REGION Network 40: [Job]Transfer P&P Left Select Job [to Hipot&Thinkness]
   // Configure here when the jobs of the sequence should be started. More jobs could be added.
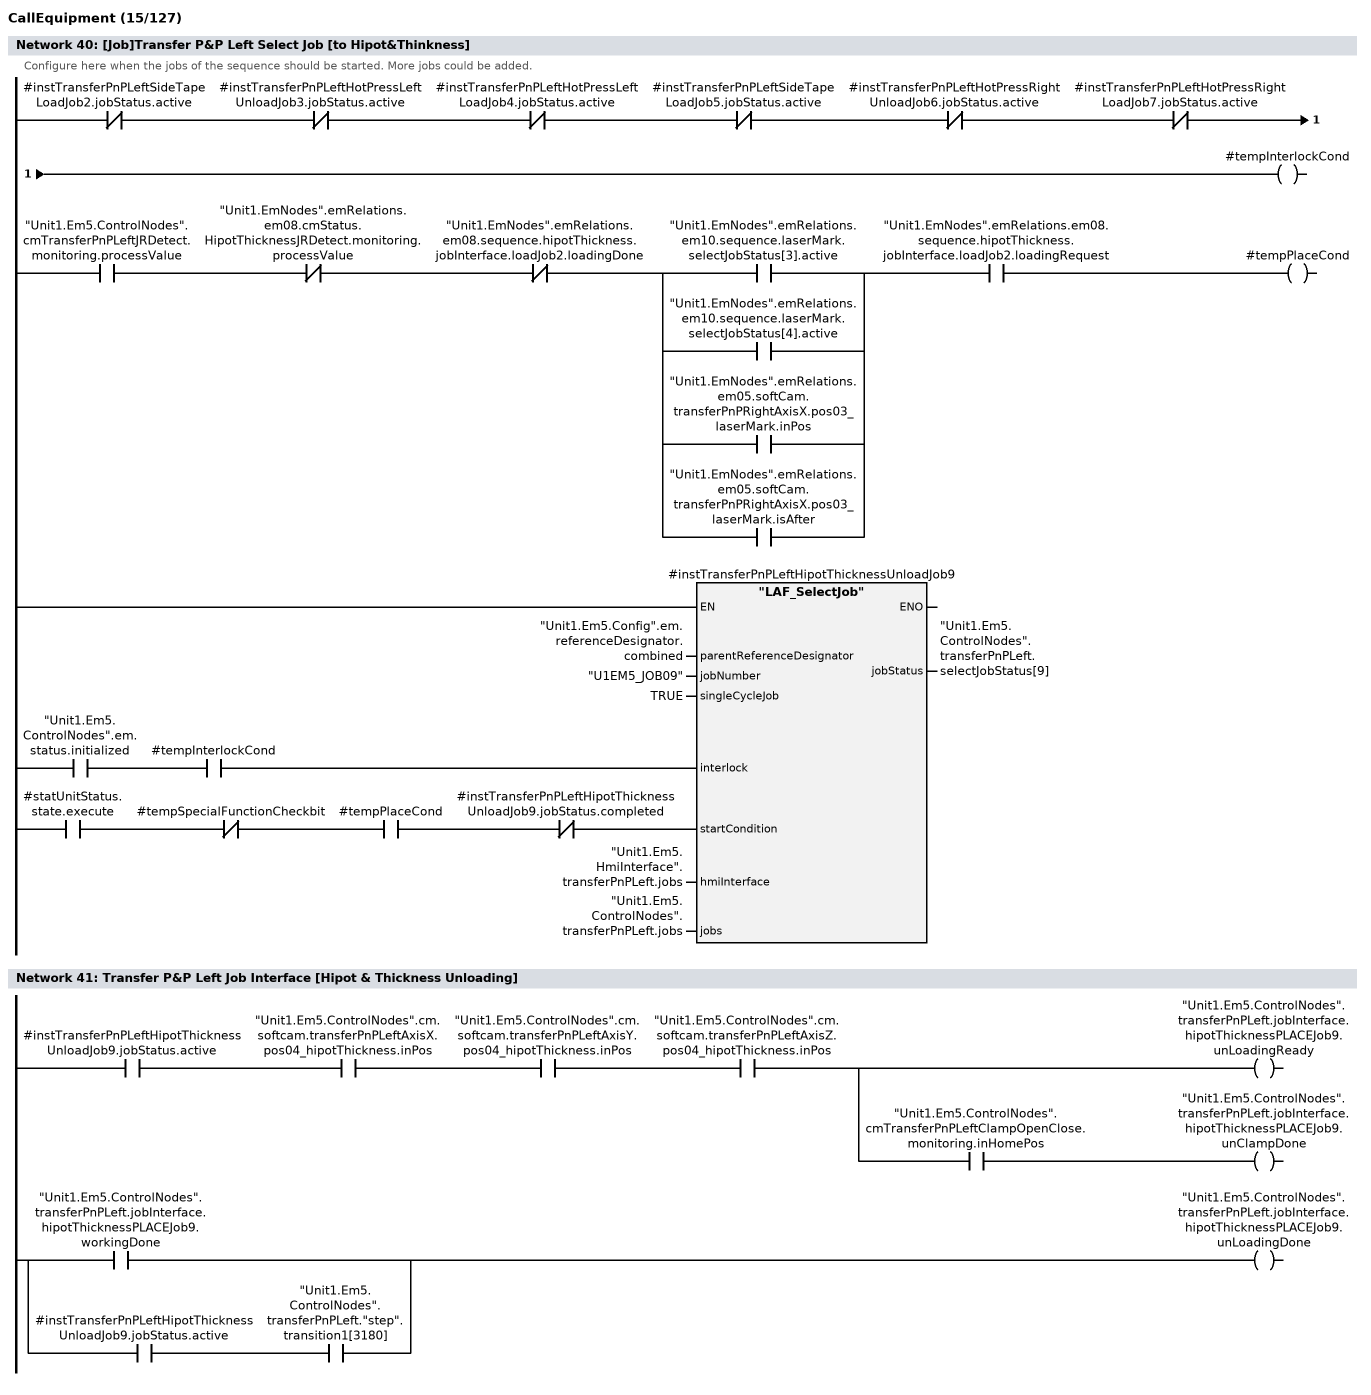
   RUNG wire#powerrail
      I_Contact( #instTransferPnPLeftSideTapeLoadJob2.jobStatus.active )
      I_Contact( #instTransferPnPLeftHotPressLeftUnloadJob3.jobStatus.active )
      I_Contact( #instTransferPnPLeftHotPressLeftLoadJob4.jobStatus.active )
      I_Contact( #instTransferPnPLeftSideTapeLoadJob5.jobStatus.active )
      I_Contact( #instTransferPnPLeftHotPressRightUnloadJob6.jobStatus.active )
      I_Contact( #instTransferPnPLeftHotPressRightLoadJob7.jobStatus.active )
      Coil( #tempInterlockCond )
   END_RUNG
   RUNG wire#powerrail
      Contact( "Unit1.Em5.ControlNodes".cmTransferPnPLeftJRDetect.monitoring.processValue )
      I_Contact( "Unit1.EmNodes".emRelations.em08.cmStatus.HipotThicknessJRDetect.monitoring.processValue )
      I_Contact( "Unit1.EmNodes".emRelations.em08.sequence.hipotThickness.jobInterface.loadJob2.loadingDone )
      wire#w1
      Contact( "Unit1.EmNodes".emRelations.em10.sequence.laserMark.selectJobStatus[3].active )
      wire#w2
      Contact( "Unit1.EmNodes".emRelations.em08.sequence.hipotThickness.jobInterface.loadJob2.loadingRequest )
      Coil( #tempPlaceCond )
   END_RUNG
   RUNG wire#w1
      Contact( "Unit1.EmNodes".emRelations.em10.sequence.laserMark.selectJobStatus[4].active )
   END_RUNG wire#w2
   RUNG wire#w1
      Contact( "Unit1.EmNodes".emRelations.em05.softCam.transferPnPRightAxisX.pos03_laserMark.inPos )
   END_RUNG wire#w2
   RUNG wire#w1
      Contact( "Unit1.EmNodes".emRelations.em05.softCam.transferPnPRightAxisX.pos03_laserMark.isAfter )
   END_RUNG wire#w2
   RUNG wire#powerrail
      #instTransferPnPLeftHipotThicknessUnloadJob9(interlock := wire#w3, startCondition := wire#w4, parentReferenceDesignator := "Unit1.Em5.Config".em.referenceDesignator.combined, jobNumber := "U1EM5_JOB09", singleCycleJob := TRUE, hmiInterface := "Unit1.Em5.HmiInterface".transferPnPLeft.jobs, jobs := "Unit1.Em5.ControlNodes".transferPnPLeft.jobs, jobStatus => "Unit1.Em5.ControlNodes".transferPnPLeft.selectJobStatus[9])
   END_RUNG
   RUNG wire#powerrail
      Contact( "Unit1.Em5.ControlNodes".em.status.initialized )
      Contact( #tempInterlockCond )
   END_RUNG wire#w3
   RUNG wire#powerrail
      Contact( #statUnitStatus.state.execute )
      I_Contact( #tempSpecialFunctionCheckbit )
      Contact( #tempPlaceCond )
      I_Contact( #instTransferPnPLeftHipotThicknessUnloadJob9.jobStatus.completed )
   END_RUNG wire#w4
   // the same network as SCL:
   #tempInterlockCond := NOT #instTransferPnPLeftSideTapeLoadJob2.jobStatus.active AND NOT #instTransferPnPLeftHotPressLeftUnloadJob3.jobStatus.active AND NOT #instTransferPnPLeftHotPressLeftLoadJob4.jobStatus.active AND NOT #instTransferPnPLeftSideTapeLoadJob5.jobStatus.active AND NOT #instTransferPnPLeftHotPressRightUnloadJob6.jobStatus.active AND NOT #instTransferPnPLeftHotPressRightLoadJob7.jobStatus.active;
   #tempPlaceCond := "Unit1.Em5.ControlNodes".cmTransferPnPLeftJRDetect.monitoring.processValue AND NOT "Unit1.EmNodes".emRelations.em08.cmStatus.HipotThicknessJRDetect.monitoring.processValue AND NOT "Unit1.EmNodes".emRelations.em08.sequence.hipotThickness.jobInterface.loadJob2.loadingDone AND ("Unit1.EmNodes".emRelations.em10.sequence.laserMark.selectJobStatus[3].active OR "Unit1.EmNodes".emRelations.em10.sequence.laserMark.selectJobStatus[4].active OR "Unit1.EmNodes".emRelations.em05.softCam.transferPnPRightAxisX.pos03_laserMark.inPos OR "Unit1.EmNodes".emRelations.em05.softCam.transferPnPRightAxisX.pos03_laserMark.isAfter) AND "Unit1.EmNodes".emRelations.em08.sequence.hipotThickness.jobInterface.loadJob2.loadingRequest;
   #instTransferPnPLeftHipotThicknessUnloadJob9(parentReferenceDesignator := "Unit1.Em5.Config".em.referenceDesignator.combined,   // "LAF_SelectJob"
                           jobNumber := "U1EM5_JOB09",
                           singleCycleJob := TRUE,
                           interlock := "Unit1.Em5.ControlNodes".em.status.initialized AND #tempInterlockCond,
                           startCondition := #statUnitStatus.state.execute AND NOT #tempSpecialFunctionCheckbit AND #tempPlaceCond AND NOT #instTransferPnPLeftHipotThicknessUnloadJob9.jobStatus.completed,
                           hmiInterface := "Unit1.Em5.HmiInterface".transferPnPLeft.jobs,
                           jobs := "Unit1.Em5.ControlNodes".transferPnPLeft.jobs,
                           jobStatus => "Unit1.Em5.ControlNodes".transferPnPLeft.selectJobStatus[9]);
END_REGION

REGION Network 41: Transfer P&P Left Job Interface [Hipot & Thickness Unloading]
   RUNG wire#powerrail
      Contact( #instTransferPnPLeftHipotThicknessUnloadJob9.jobStatus.active )
      Contact( "Unit1.Em5.ControlNodes".cm.softcam.transferPnPLeftAxisX.pos04_hipotThickness.inPos )
      Contact( "Unit1.Em5.ControlNodes".cm.softcam.transferPnPLeftAxisY.pos04_hipotThickness.inPos )
      Contact( "Unit1.Em5.ControlNodes".cm.softcam.transferPnPLeftAxisZ.pos04_hipotThickness.inPos )
      wire#w1
      Coil( "Unit1.Em5.ControlNodes".transferPnPLeft.jobInterface.hipotThicknessPLACEJob9.unLoadingReady )
   END_RUNG
   RUNG wire#w1
      Contact( "Unit1.Em5.ControlNodes".cmTransferPnPLeftClampOpenClose.monitoring.inHomePos )
      Coil( "Unit1.Em5.ControlNodes".transferPnPLeft.jobInterface.hipotThicknessPLACEJob9.unClampDone )
   END_RUNG
   RUNG wire#powerrail
      Contact( "Unit1.Em5.ControlNodes".transferPnPLeft.jobInterface.hipotThicknessPLACEJob9.workingDone )
      wire#w2
      Coil( "Unit1.Em5.ControlNodes".transferPnPLeft.jobInterface.hipotThicknessPLACEJob9.unLoadingDone )
   END_RUNG
   RUNG wire#powerrail
      Contact( #instTransferPnPLeftHipotThicknessUnloadJob9.jobStatus.active )
      Contact( "Unit1.Em5.ControlNodes".transferPnPLeft."step".transition1[3180] )
   END_RUNG wire#w2
   // the same network as SCL:
   "Unit1.Em5.ControlNodes".transferPnPLeft.jobInterface.hipotThicknessPLACEJob9.unLoadingReady := #instTransferPnPLeftHipotThicknessUnloadJob9.jobStatus.active AND "Unit1.Em5.ControlNodes".cm.softcam.transferPnPLeftAxisX.pos04_hipotThickness.inPos AND "Unit1.Em5.ControlNodes".cm.softcam.transferPnPLeftAxisY.pos04_hipotThickness.inPos AND "Unit1.Em5.ControlNodes".cm.softcam.transferPnPLeftAxisZ.pos04_hipotThickness.inPos;
   "Unit1.Em5.ControlNodes".transferPnPLeft.jobInterface.hipotThicknessPLACEJob9.unClampDone := "Unit1.Em5.ControlNodes".transferPnPLeft.jobInterface.hipotThicknessPLACEJob9.unLoadingReady AND "Unit1.Em5.ControlNodes".cmTransferPnPLeftClampOpenClose.monitoring.inHomePos;
   "Unit1.Em5.ControlNodes".transferPnPLeft.jobInterface.hipotThicknessPLACEJob9.unLoadingDone := "Unit1.Em5.ControlNodes".transferPnPLeft.jobInterface.hipotThicknessPLACEJob9.workingDone OR (#instTransferPnPLeftHipotThicknessUnloadJob9.jobStatus.active AND "Unit1.Em5.ControlNodes".transferPnPLeft."step".transition1[3180]);
END_REGION

REGION Network 42: Transfer P&P Left Job Interface Working Done [HotPress Left/Right → Hipot&Thickness]
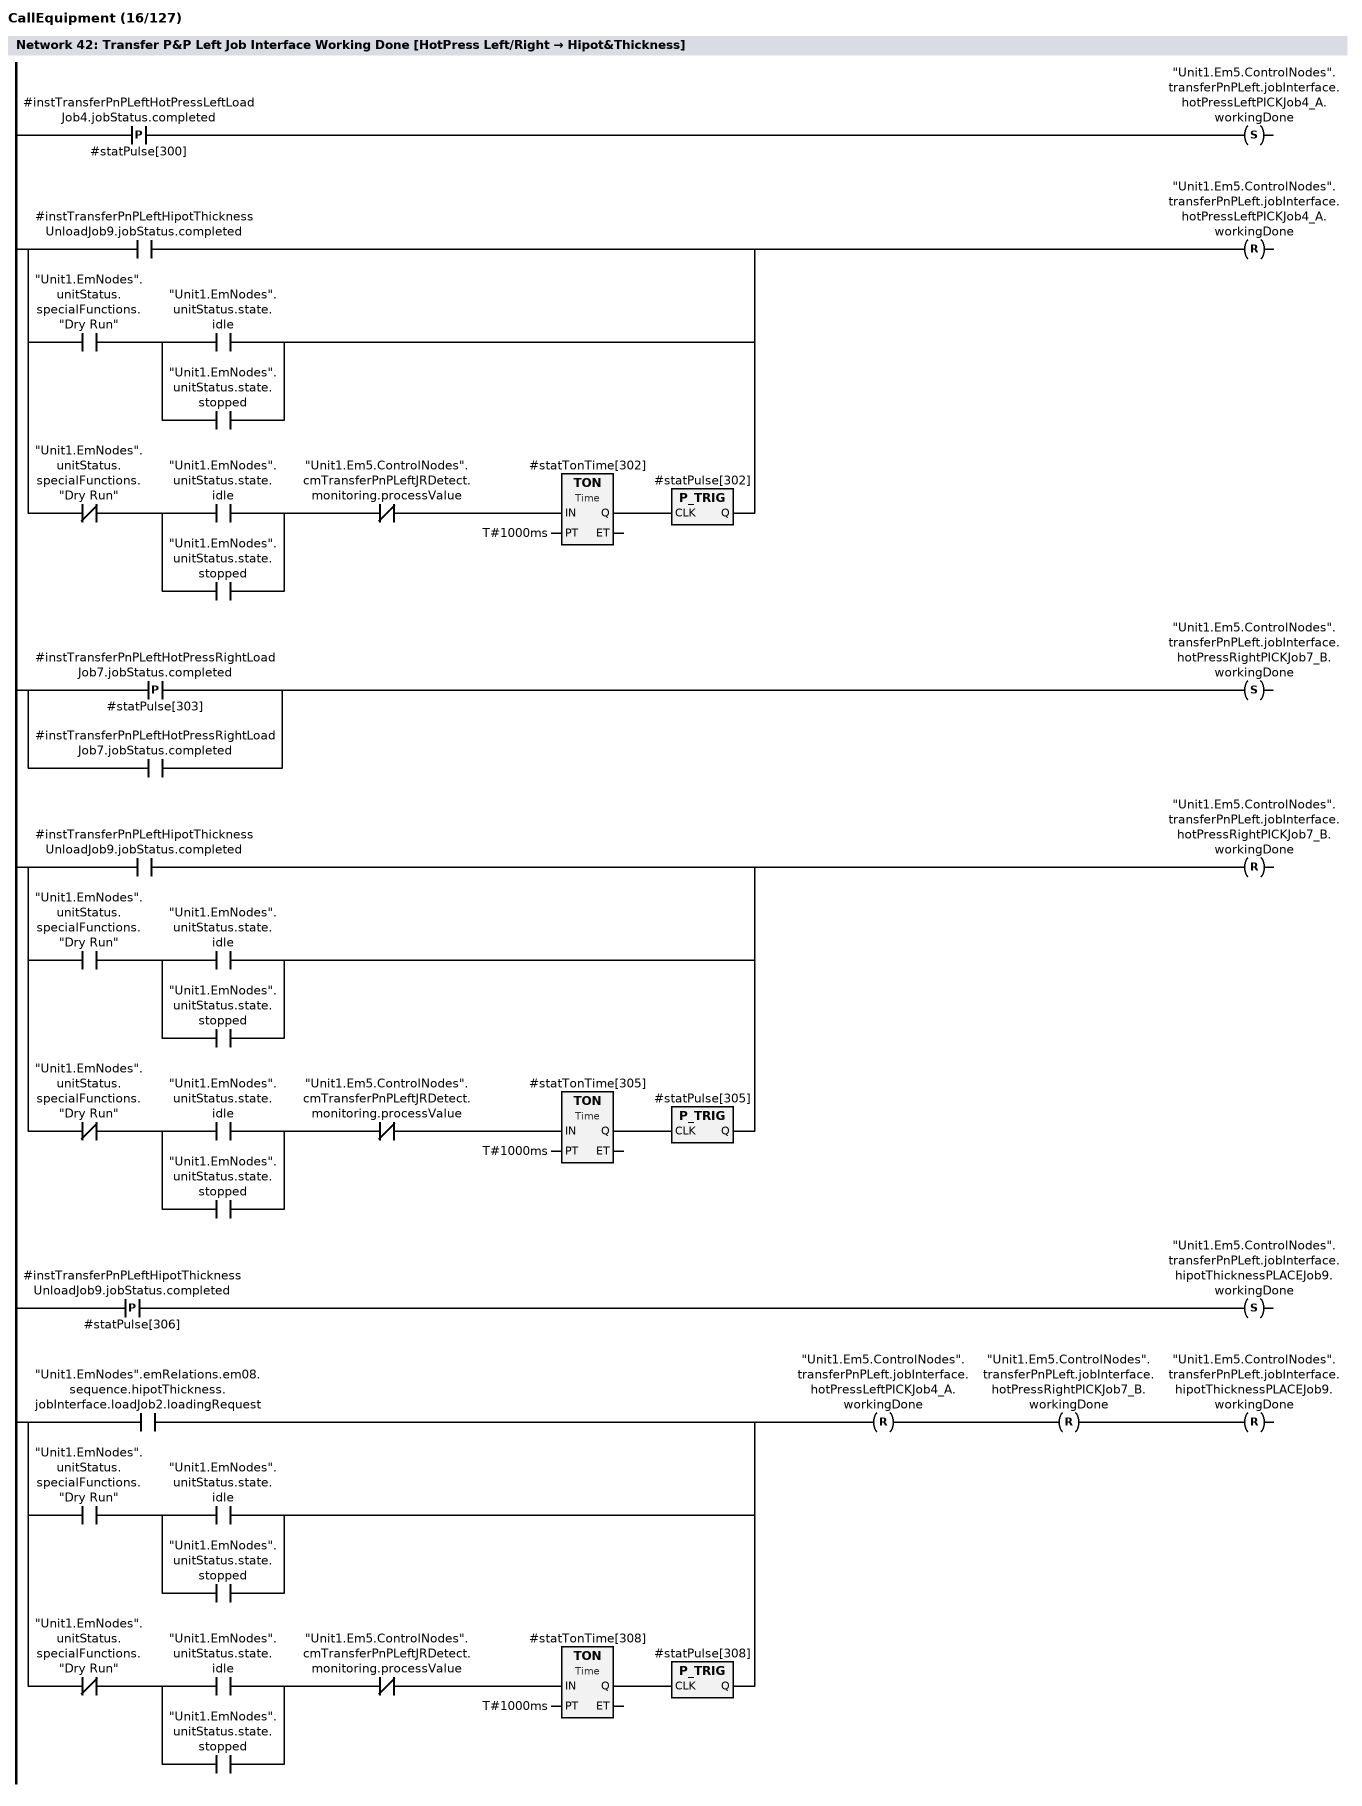
   RUNG wire#powerrail
      P_Contact(operand := #instTransferPnPLeftHotPressLeftLoadJob4.jobStatus.completed, bit := #statPulse[300])
      S_Coil( "Unit1.Em5.ControlNodes".transferPnPLeft.jobInterface.hotPressLeftPICKJob4_A.workingDone )
   END_RUNG
   RUNG wire#powerrail
      Contact( #instTransferPnPLeftHipotThicknessUnloadJob9.jobStatus.completed )
      wire#w1
      R_Coil( "Unit1.Em5.ControlNodes".transferPnPLeft.jobInterface.hotPressLeftPICKJob4_A.workingDone )
   END_RUNG
   RUNG wire#powerrail
      Contact( "Unit1.EmNodes".unitStatus.specialFunctions."Dry Run" )
      wire#w2
      Contact( "Unit1.EmNodes".unitStatus.state.idle )
   END_RUNG wire#w1
   RUNG wire#w2
      Contact( "Unit1.EmNodes".unitStatus.state.stopped )
   END_RUNG wire#w1
   RUNG wire#powerrail
      I_Contact( "Unit1.EmNodes".unitStatus.specialFunctions."Dry Run" )
      wire#w3
      Contact( "Unit1.EmNodes".unitStatus.state.idle )
      wire#w4
      I_Contact( "Unit1.Em5.ControlNodes".cmTransferPnPLeftJRDetect.monitoring.processValue )
      { S7_Templates := "time_type := Time" } #statTonTime[302].TON(pt := T#1000ms, et =>)
      P_Trig( #statPulse[302] )
   END_RUNG wire#w1
   RUNG wire#w3
      Contact( "Unit1.EmNodes".unitStatus.state.stopped )
   END_RUNG wire#w4
   RUNG wire#powerrail
      P_Contact(operand := #instTransferPnPLeftHotPressRightLoadJob7.jobStatus.completed, bit := #statPulse[303])
      wire#w5
      S_Coil( "Unit1.Em5.ControlNodes".transferPnPLeft.jobInterface.hotPressRightPICKJob7_B.workingDone )
   END_RUNG
   RUNG wire#powerrail
      Contact( #instTransferPnPLeftHotPressRightLoadJob7.jobStatus.completed )
   END_RUNG wire#w5
   RUNG wire#powerrail
      Contact( #instTransferPnPLeftHipotThicknessUnloadJob9.jobStatus.completed )
      wire#w6
      R_Coil( "Unit1.Em5.ControlNodes".transferPnPLeft.jobInterface.hotPressRightPICKJob7_B.workingDone )
   END_RUNG
   RUNG wire#powerrail
      Contact( "Unit1.EmNodes".unitStatus.specialFunctions."Dry Run" )
      wire#w7
      Contact( "Unit1.EmNodes".unitStatus.state.idle )
   END_RUNG wire#w6
   RUNG wire#w7
      Contact( "Unit1.EmNodes".unitStatus.state.stopped )
   END_RUNG wire#w6
   RUNG wire#powerrail
      I_Contact( "Unit1.EmNodes".unitStatus.specialFunctions."Dry Run" )
      wire#w8
      Contact( "Unit1.EmNodes".unitStatus.state.idle )
      wire#w9
      I_Contact( "Unit1.Em5.ControlNodes".cmTransferPnPLeftJRDetect.monitoring.processValue )
      { S7_Templates := "time_type := Time" } #statTonTime[305].TON(pt := T#1000ms, et =>)
      P_Trig( #statPulse[305] )
   END_RUNG wire#w6
   RUNG wire#w8
      Contact( "Unit1.EmNodes".unitStatus.state.stopped )
   END_RUNG wire#w9
   RUNG wire#powerrail
      P_Contact(operand := #instTransferPnPLeftHipotThicknessUnloadJob9.jobStatus.completed, bit := #statPulse[306])
      S_Coil( "Unit1.Em5.ControlNodes".transferPnPLeft.jobInterface.hipotThicknessPLACEJob9.workingDone )
   END_RUNG
   RUNG wire#powerrail
      Contact( "Unit1.EmNodes".emRelations.em08.sequence.hipotThickness.jobInterface.loadJob2.loadingRequest )
      wire#w10
      R_Coil( "Unit1.Em5.ControlNodes".transferPnPLeft.jobInterface.hotPressLeftPICKJob4_A.workingDone )
      R_Coil( "Unit1.Em5.ControlNodes".transferPnPLeft.jobInterface.hotPressRightPICKJob7_B.workingDone )
      R_Coil( "Unit1.Em5.ControlNodes".transferPnPLeft.jobInterface.hipotThicknessPLACEJob9.workingDone )
   END_RUNG
   RUNG wire#powerrail
      Contact( "Unit1.EmNodes".unitStatus.specialFunctions."Dry Run" )
      wire#w11
      Contact( "Unit1.EmNodes".unitStatus.state.idle )
   END_RUNG wire#w10
   RUNG wire#w11
      Contact( "Unit1.EmNodes".unitStatus.state.stopped )
   END_RUNG wire#w10
   RUNG wire#powerrail
      I_Contact( "Unit1.EmNodes".unitStatus.specialFunctions."Dry Run" )
      wire#w12
      Contact( "Unit1.EmNodes".unitStatus.state.idle )
      wire#w13
      I_Contact( "Unit1.Em5.ControlNodes".cmTransferPnPLeftJRDetect.monitoring.processValue )
      { S7_Templates := "time_type := Time" } #statTonTime[308].TON(pt := T#1000ms, et =>)
      P_Trig( #statPulse[308] )
   END_RUNG wire#w10
   RUNG wire#w12
      Contact( "Unit1.EmNodes".unitStatus.state.stopped )
   END_RUNG wire#w13
   // the same network as SCL:
   #_w1 := #instTransferPnPLeftHotPressLeftLoadJob4.jobStatus.completed AND NOT #statPulse[300];   // rising edge of #instTransferPnPLeftHotPressLeftLoadJob4.jobStatus.completed
   #statPulse[300] := #instTransferPnPLeftHotPressLeftLoadJob4.jobStatus.completed;
   IF #_w1 THEN
       "Unit1.Em5.ControlNodes".transferPnPLeft.jobInterface.hotPressLeftPICKJob4_A.workingDone := TRUE;
   END_IF;
   #statTonTime[302].TON(IN := NOT "Unit1.EmNodes".unitStatus.specialFunctions."Dry Run" AND ("Unit1.EmNodes".unitStatus.state.idle OR "Unit1.EmNodes".unitStatus.state.stopped) AND NOT "Unit1.Em5.ControlNodes".cmTransferPnPLeftJRDetect.monitoring.processValue,
                         PT := T#1000ms);
   #_w2 := #statTonTime[302].Q AND NOT #statPulse[302];   // rising edge
   #statPulse[302] := #statTonTime[302].Q;
   IF #instTransferPnPLeftHipotThicknessUnloadJob9.jobStatus.completed OR ("Unit1.EmNodes".unitStatus.specialFunctions."Dry Run" AND ("Unit1.EmNodes".unitStatus.state.idle OR "Unit1.EmNodes".unitStatus.state.stopped)) OR #_w2 THEN
       "Unit1.Em5.ControlNodes".transferPnPLeft.jobInterface.hotPressLeftPICKJob4_A.workingDone := FALSE;
   END_IF;
   #_w3 := #instTransferPnPLeftHotPressRightLoadJob7.jobStatus.completed AND NOT #statPulse[303];   // rising edge of #instTransferPnPLeftHotPressRightLoadJob7.jobStatus.completed
   #statPulse[303] := #instTransferPnPLeftHotPressRightLoadJob7.jobStatus.completed;
   IF #_w3 OR #instTransferPnPLeftHotPressRightLoadJob7.jobStatus.completed THEN
       "Unit1.Em5.ControlNodes".transferPnPLeft.jobInterface.hotPressRightPICKJob7_B.workingDone := TRUE;
   END_IF;
   #statTonTime[305].TON(IN := NOT "Unit1.EmNodes".unitStatus.specialFunctions."Dry Run" AND ("Unit1.EmNodes".unitStatus.state.idle OR "Unit1.EmNodes".unitStatus.state.stopped) AND NOT "Unit1.Em5.ControlNodes".cmTransferPnPLeftJRDetect.monitoring.processValue,
                         PT := T#1000ms);
   #_w4 := #statTonTime[305].Q AND NOT #statPulse[305];   // rising edge
   #statPulse[305] := #statTonTime[305].Q;
   IF #instTransferPnPLeftHipotThicknessUnloadJob9.jobStatus.completed OR ("Unit1.EmNodes".unitStatus.specialFunctions."Dry Run" AND ("Unit1.EmNodes".unitStatus.state.idle OR "Unit1.EmNodes".unitStatus.state.stopped)) OR #_w4 THEN
       "Unit1.Em5.ControlNodes".transferPnPLeft.jobInterface.hotPressRightPICKJob7_B.workingDone := FALSE;
   END_IF;
   #_w5 := #instTransferPnPLeftHipotThicknessUnloadJob9.jobStatus.completed AND NOT #statPulse[306];   // rising edge of #instTransferPnPLeftHipotThicknessUnloadJob9.jobStatus.completed
   #statPulse[306] := #instTransferPnPLeftHipotThicknessUnloadJob9.jobStatus.completed;
   IF #_w5 THEN
       "Unit1.Em5.ControlNodes".transferPnPLeft.jobInterface.hipotThicknessPLACEJob9.workingDone := TRUE;
   END_IF;
   #statTonTime[308].TON(IN := NOT "Unit1.EmNodes".unitStatus.specialFunctions."Dry Run" AND ("Unit1.EmNodes".unitStatus.state.idle OR "Unit1.EmNodes".unitStatus.state.stopped) AND NOT "Unit1.Em5.ControlNodes".cmTransferPnPLeftJRDetect.monitoring.processValue,
                         PT := T#1000ms);
   #_w6 := #statTonTime[308].Q AND NOT #statPulse[308];   // rising edge
   #statPulse[308] := #statTonTime[308].Q;
   IF "Unit1.EmNodes".emRelations.em08.sequence.hipotThickness.jobInterface.loadJob2.loadingRequest OR ("Unit1.EmNodes".unitStatus.specialFunctions."Dry Run" AND ("Unit1.EmNodes".unitStatus.state.idle OR "Unit1.EmNodes".unitStatus.state.stopped)) OR #_w6 THEN
       "Unit1.Em5.ControlNodes".transferPnPLeft.jobInterface.hotPressLeftPICKJob4_A.workingDone := FALSE;
       "Unit1.Em5.ControlNodes".transferPnPLeft.jobInterface.hotPressRightPICKJob7_B.workingDone := FALSE;
       "Unit1.Em5.ControlNodes".transferPnPLeft.jobInterface.hipotThicknessPLACEJob9.workingDone := FALSE;
   END_IF;
END_REGION

REGION Network 44: [Condition] Transfer P&P Right Job
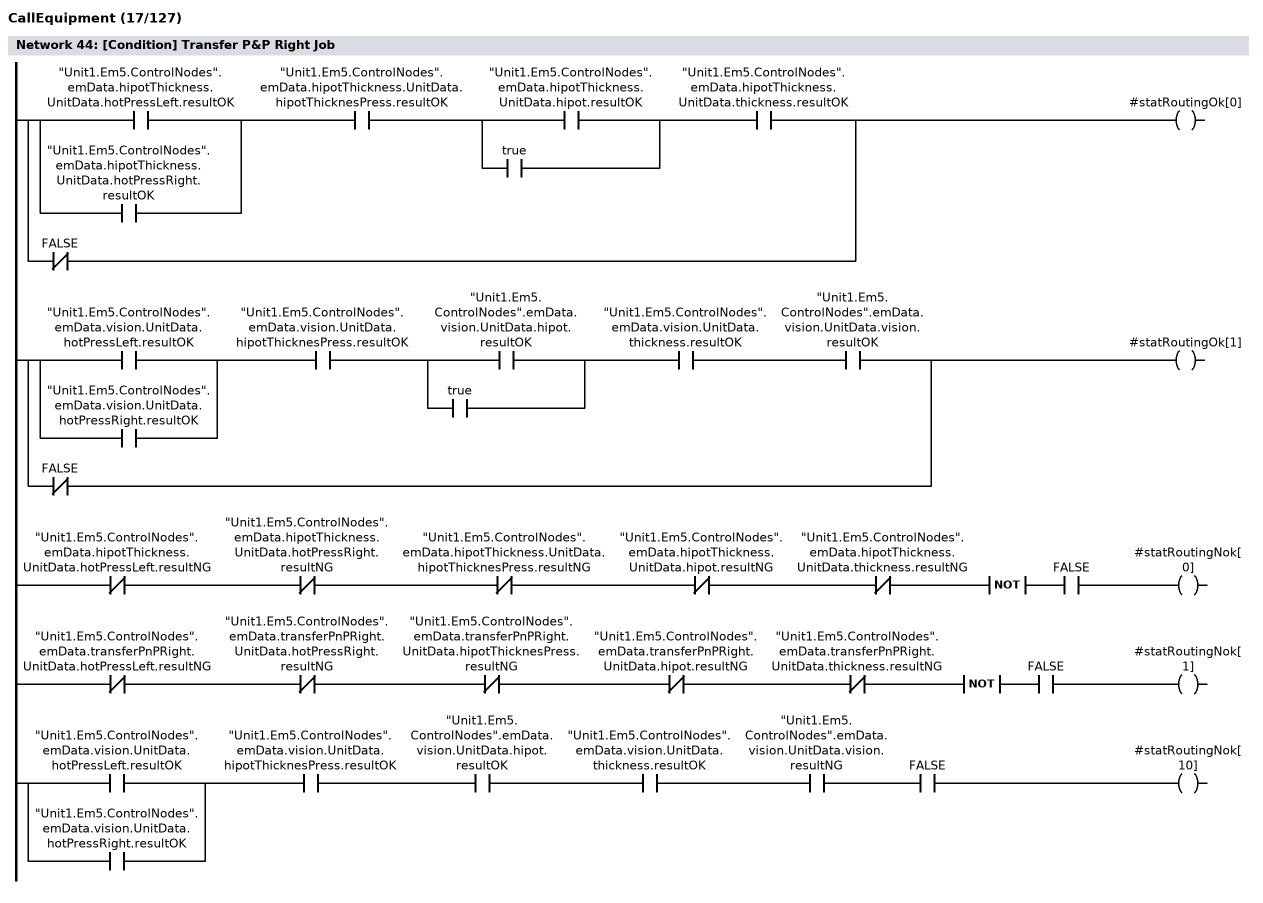
   RUNG wire#powerrail
      Contact( "Unit1.Em5.ControlNodes".emData.hipotThickness.UnitData.hotPressLeft.resultOK )
      wire#w1
      Contact( "Unit1.Em5.ControlNodes".emData.hipotThickness.UnitData.hipotThicknesPress.resultOK )
      wire#w2
      Contact( "Unit1.Em5.ControlNodes".emData.hipotThickness.UnitData.hipot.resultOK )
      wire#w3
      Contact( "Unit1.Em5.ControlNodes".emData.hipotThickness.UnitData.thickness.resultOK )
      wire#w4
      Coil( #statRoutingOk[0] )
   END_RUNG
   RUNG wire#powerrail
      Contact( "Unit1.Em5.ControlNodes".emData.hipotThickness.UnitData.hotPressRight.resultOK )
   END_RUNG wire#w1
   RUNG wire#w2
      Contact( true )
   END_RUNG wire#w3
   RUNG wire#powerrail
      I_Contact( FALSE )
   END_RUNG wire#w4
   RUNG wire#powerrail
      Contact( "Unit1.Em5.ControlNodes".emData.vision.UnitData.hotPressLeft.resultOK )
      wire#w5
      Contact( "Unit1.Em5.ControlNodes".emData.vision.UnitData.hipotThicknesPress.resultOK )
      wire#w6
      Contact( "Unit1.Em5.ControlNodes".emData.vision.UnitData.hipot.resultOK )
      wire#w7
      Contact( "Unit1.Em5.ControlNodes".emData.vision.UnitData.thickness.resultOK )
      Contact( "Unit1.Em5.ControlNodes".emData.vision.UnitData.vision.resultOK )
      wire#w8
      Coil( #statRoutingOk[1] )
   END_RUNG
   RUNG wire#powerrail
      Contact( "Unit1.Em5.ControlNodes".emData.vision.UnitData.hotPressRight.resultOK )
   END_RUNG wire#w5
   RUNG wire#w6
      Contact( true )
   END_RUNG wire#w7
   RUNG wire#powerrail
      I_Contact( FALSE )
   END_RUNG wire#w8
   RUNG wire#powerrail
      I_Contact( "Unit1.Em5.ControlNodes".emData.hipotThickness.UnitData.hotPressLeft.resultNG )
      I_Contact( "Unit1.Em5.ControlNodes".emData.hipotThickness.UnitData.hotPressRight.resultNG )
      I_Contact( "Unit1.Em5.ControlNodes".emData.hipotThickness.UnitData.hipotThicknesPress.resultNG )
      I_Contact( "Unit1.Em5.ControlNodes".emData.hipotThickness.UnitData.hipot.resultNG )
      I_Contact( "Unit1.Em5.ControlNodes".emData.hipotThickness.UnitData.thickness.resultNG )
      Not()
      Contact( FALSE )
      Coil( #statRoutingNok[0] )
   END_RUNG
   RUNG wire#powerrail
      I_Contact( "Unit1.Em5.ControlNodes".emData.transferPnPRight.UnitData.hotPressLeft.resultNG )
      I_Contact( "Unit1.Em5.ControlNodes".emData.transferPnPRight.UnitData.hotPressRight.resultNG )
      I_Contact( "Unit1.Em5.ControlNodes".emData.transferPnPRight.UnitData.hipotThicknesPress.resultNG )
      I_Contact( "Unit1.Em5.ControlNodes".emData.transferPnPRight.UnitData.hipot.resultNG )
      I_Contact( "Unit1.Em5.ControlNodes".emData.transferPnPRight.UnitData.thickness.resultNG )
      Not()
      Contact( FALSE )
      Coil( #statRoutingNok[1] )
   END_RUNG
   RUNG wire#powerrail
      Contact( "Unit1.Em5.ControlNodes".emData.vision.UnitData.hotPressLeft.resultOK )
      wire#w9
      Contact( "Unit1.Em5.ControlNodes".emData.vision.UnitData.hipotThicknesPress.resultOK )
      Contact( "Unit1.Em5.ControlNodes".emData.vision.UnitData.hipot.resultOK )
      Contact( "Unit1.Em5.ControlNodes".emData.vision.UnitData.thickness.resultOK )
      Contact( "Unit1.Em5.ControlNodes".emData.vision.UnitData.vision.resultNG )
      Contact( FALSE )
      Coil( #statRoutingNok[10] )
   END_RUNG
   RUNG wire#powerrail
      Contact( "Unit1.Em5.ControlNodes".emData.vision.UnitData.hotPressRight.resultOK )
   END_RUNG wire#w9
   // the same network as SCL:
   #statRoutingOk[0] := (("Unit1.Em5.ControlNodes".emData.hipotThickness.UnitData.hotPressLeft.resultOK OR "Unit1.Em5.ControlNodes".emData.hipotThickness.UnitData.hotPressRight.resultOK) AND "Unit1.Em5.ControlNodes".emData.hipotThickness.UnitData.hipotThicknesPress.resultOK AND ("Unit1.Em5.ControlNodes".emData.hipotThickness.UnitData.hipot.resultOK OR true) AND "Unit1.Em5.ControlNodes".emData.hipotThickness.UnitData.thickness.resultOK) OR NOT FALSE;
   #statRoutingOk[1] := (("Unit1.Em5.ControlNodes".emData.vision.UnitData.hotPressLeft.resultOK OR "Unit1.Em5.ControlNodes".emData.vision.UnitData.hotPressRight.resultOK) AND "Unit1.Em5.ControlNodes".emData.vision.UnitData.hipotThicknesPress.resultOK AND ("Unit1.Em5.ControlNodes".emData.vision.UnitData.hipot.resultOK OR true) AND "Unit1.Em5.ControlNodes".emData.vision.UnitData.thickness.resultOK AND "Unit1.Em5.ControlNodes".emData.vision.UnitData.vision.resultOK) OR NOT FALSE;
   #statRoutingNok[0] := NOT (NOT "Unit1.Em5.ControlNodes".emData.hipotThickness.UnitData.hotPressLeft.resultNG AND NOT "Unit1.Em5.ControlNodes".emData.hipotThickness.UnitData.hotPressRight.resultNG AND NOT "Unit1.Em5.ControlNodes".emData.hipotThickness.UnitData.hipotThicknesPress.resultNG AND NOT "Unit1.Em5.ControlNodes".emData.hipotThickness.UnitData.hipot.resultNG AND NOT "Unit1.Em5.ControlNodes".emData.hipotThickness.UnitData.thickness.resultNG) AND FALSE;
   #statRoutingNok[1] := NOT (NOT "Unit1.Em5.ControlNodes".emData.transferPnPRight.UnitData.hotPressLeft.resultNG AND NOT "Unit1.Em5.ControlNodes".emData.transferPnPRight.UnitData.hotPressRight.resultNG AND NOT "Unit1.Em5.ControlNodes".emData.transferPnPRight.UnitData.hipotThicknesPress.resultNG AND NOT "Unit1.Em5.ControlNodes".emData.transferPnPRight.UnitData.hipot.resultNG AND NOT "Unit1.Em5.ControlNodes".emData.transferPnPRight.UnitData.thickness.resultNG) AND FALSE;
   #statRoutingNok[10] := ("Unit1.Em5.ControlNodes".emData.vision.UnitData.hotPressLeft.resultOK OR "Unit1.Em5.ControlNodes".emData.vision.UnitData.hotPressRight.resultOK) AND "Unit1.Em5.ControlNodes".emData.vision.UnitData.hipotThicknesPress.resultOK AND "Unit1.Em5.ControlNodes".emData.vision.UnitData.hipot.resultOK AND "Unit1.Em5.ControlNodes".emData.vision.UnitData.thickness.resultOK AND "Unit1.Em5.ControlNodes".emData.vision.UnitData.vision.resultNG AND FALSE;
END_REGION

REGION Network 45: [Job] Transfer P&P Right Select Job [initializing]
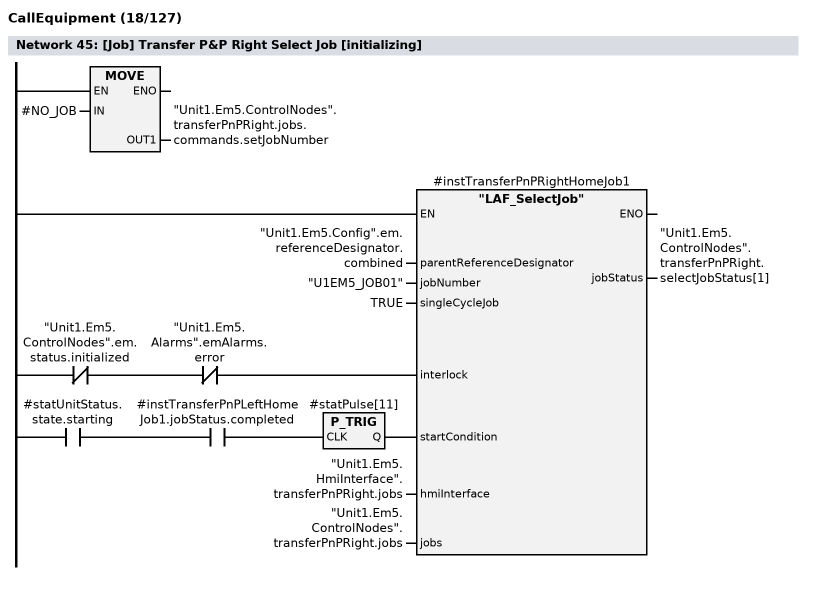
   RUNG wire#powerrail
      Move(in := #NO_JOB, out1 => "Unit1.Em5.ControlNodes".transferPnPRight.jobs.commands.setJobNumber)
   END_RUNG
   RUNG wire#powerrail
      #instTransferPnPRightHomeJob1(interlock := wire#w1, startCondition := wire#w2, parentReferenceDesignator := "Unit1.Em5.Config".em.referenceDesignator.combined, jobNumber := "U1EM5_JOB01", singleCycleJob := TRUE, hmiInterface := "Unit1.Em5.HmiInterface".transferPnPRight.jobs, jobs := "Unit1.Em5.ControlNodes".transferPnPRight.jobs, jobStatus => "Unit1.Em5.ControlNodes".transferPnPRight.selectJobStatus[1])
   END_RUNG
   RUNG wire#powerrail
      I_Contact( "Unit1.Em5.ControlNodes".em.status.initialized )
      I_Contact( "Unit1.Em5.Alarms".emAlarms.error )
   END_RUNG wire#w1
   RUNG wire#powerrail
      Contact( #statUnitStatus.state.starting )
      Contact( #instTransferPnPLeftHomeJob1.jobStatus.completed )
      P_Trig( #statPulse[11] )
   END_RUNG wire#w2
   // the same network as SCL:
   "Unit1.Em5.ControlNodes".transferPnPRight.jobs.commands.setJobNumber := #NO_JOB;
   #_w1 := #statUnitStatus.state.starting AND #instTransferPnPLeftHomeJob1.jobStatus.completed;
   #_w2 := #_w1 AND NOT #statPulse[11];   // rising edge
   #statPulse[11] := #_w1;
   #instTransferPnPRightHomeJob1(parentReferenceDesignator := "Unit1.Em5.Config".em.referenceDesignator.combined,   // "LAF_SelectJob"
                           jobNumber := "U1EM5_JOB01",
                           singleCycleJob := TRUE,
                           interlock := NOT "Unit1.Em5.ControlNodes".em.status.initialized AND NOT "Unit1.Em5.Alarms".emAlarms.error,
                           startCondition := #_w2,
                           hmiInterface := "Unit1.Em5.HmiInterface".transferPnPRight.jobs,
                           jobs := "Unit1.Em5.ControlNodes".transferPnPRight.jobs,
                           jobStatus => "Unit1.Em5.ControlNodes".transferPnPRight.selectJobStatus[1]);
END_REGION

REGION Network 46: [Job] Transfer P&P Right Select Job
   // Configure here when the jobs of the sequence should be started. More jobs could be added.
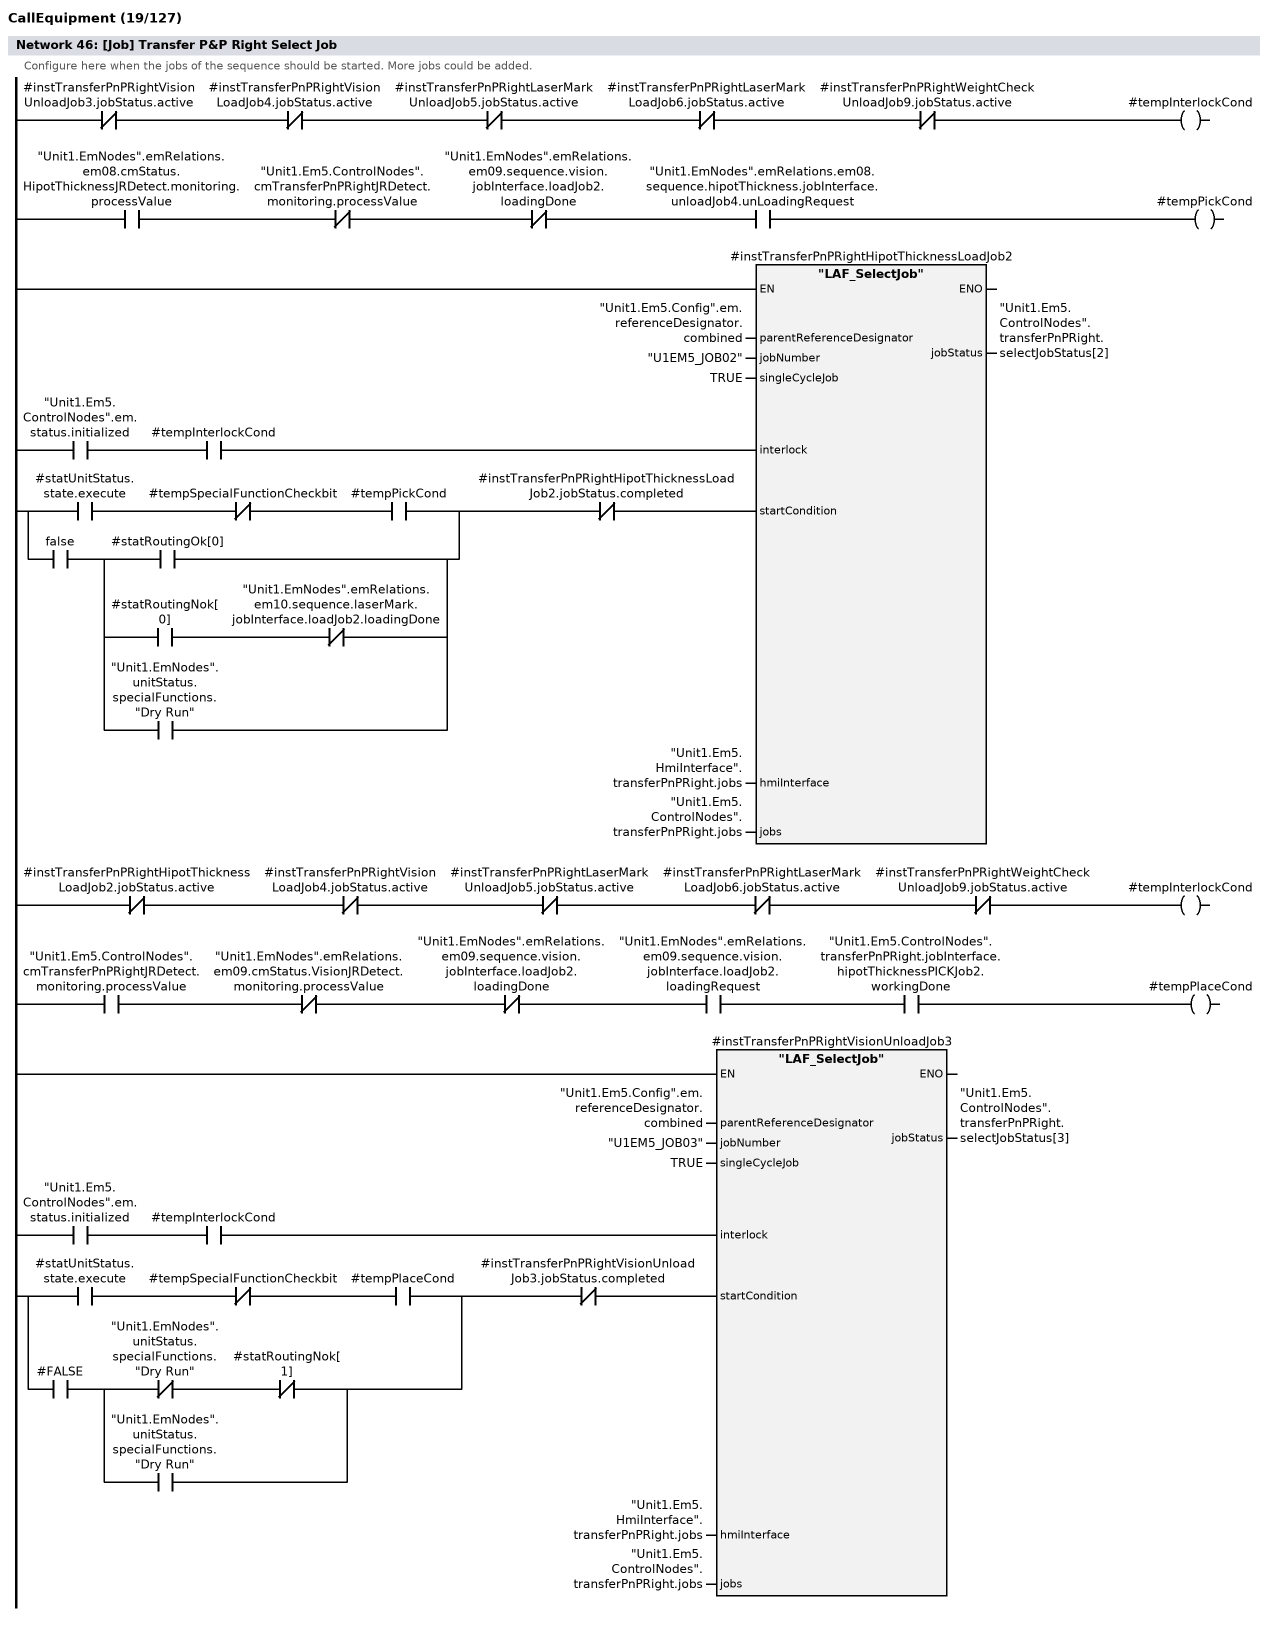
   RUNG wire#powerrail
      I_Contact( #instTransferPnPRightVisionUnloadJob3.jobStatus.active )
      I_Contact( #instTransferPnPRightVisionLoadJob4.jobStatus.active )
      I_Contact( #instTransferPnPRightLaserMarkUnloadJob5.jobStatus.active )
      I_Contact( #instTransferPnPRightLaserMarkLoadJob6.jobStatus.active )
      I_Contact( #instTransferPnPRightWeightCheckUnloadJob9.jobStatus.active )
      Coil( #tempInterlockCond )
   END_RUNG
   RUNG wire#powerrail
      Contact( "Unit1.EmNodes".emRelations.em08.cmStatus.HipotThicknessJRDetect.monitoring.processValue )
      I_Contact( "Unit1.Em5.ControlNodes".cmTransferPnPRightJRDetect.monitoring.processValue )
      I_Contact( "Unit1.EmNodes".emRelations.em09.sequence.vision.jobInterface.loadJob2.loadingDone )
      Contact( "Unit1.EmNodes".emRelations.em08.sequence.hipotThickness.jobInterface.unloadJob4.unLoadingRequest )
      Coil( #tempPickCond )
   END_RUNG
   RUNG wire#powerrail
      #instTransferPnPRightHipotThicknessLoadJob2(interlock := wire#w1, startCondition := wire#w4, parentReferenceDesignator := "Unit1.Em5.Config".em.referenceDesignator.combined, jobNumber := "U1EM5_JOB02", singleCycleJob := TRUE, hmiInterface := "Unit1.Em5.HmiInterface".transferPnPRight.jobs, jobs := "Unit1.Em5.ControlNodes".transferPnPRight.jobs, jobStatus => "Unit1.Em5.ControlNodes".transferPnPRight.selectJobStatus[2])
   END_RUNG
   RUNG wire#powerrail
      Contact( "Unit1.Em5.ControlNodes".em.status.initialized )
      Contact( #tempInterlockCond )
   END_RUNG wire#w1
   RUNG wire#powerrail
      Contact( #statUnitStatus.state.execute )
      I_Contact( #tempSpecialFunctionCheckbit )
      Contact( #tempPickCond )
      wire#w2
      I_Contact( #instTransferPnPRightHipotThicknessLoadJob2.jobStatus.completed )
   END_RUNG wire#w4
   RUNG wire#powerrail
      Contact( false )
      wire#w3
      Contact( #statRoutingOk[0] )
   END_RUNG wire#w2
   RUNG wire#w3
      Contact( #statRoutingNok[0] )
      I_Contact( "Unit1.EmNodes".emRelations.em10.sequence.laserMark.jobInterface.loadJob2.loadingDone )
   END_RUNG wire#w2
   RUNG wire#w3
      Contact( "Unit1.EmNodes".unitStatus.specialFunctions."Dry Run" )
   END_RUNG wire#w2
   RUNG wire#powerrail
      I_Contact( #instTransferPnPRightHipotThicknessLoadJob2.jobStatus.active )
      I_Contact( #instTransferPnPRightVisionLoadJob4.jobStatus.active )
      I_Contact( #instTransferPnPRightLaserMarkUnloadJob5.jobStatus.active )
      I_Contact( #instTransferPnPRightLaserMarkLoadJob6.jobStatus.active )
      I_Contact( #instTransferPnPRightWeightCheckUnloadJob9.jobStatus.active )
      Coil( #tempInterlockCond )
   END_RUNG
   RUNG wire#powerrail
      Contact( "Unit1.Em5.ControlNodes".cmTransferPnPRightJRDetect.monitoring.processValue )
      I_Contact( "Unit1.EmNodes".emRelations.em09.cmStatus.VisionJRDetect.monitoring.processValue )
      I_Contact( "Unit1.EmNodes".emRelations.em09.sequence.vision.jobInterface.loadJob2.loadingDone )
      Contact( "Unit1.EmNodes".emRelations.em09.sequence.vision.jobInterface.loadJob2.loadingRequest )
      Contact( "Unit1.Em5.ControlNodes".transferPnPRight.jobInterface.hipotThicknessPICKJob2.workingDone )
      Coil( #tempPlaceCond )
   END_RUNG
   RUNG wire#powerrail
      #instTransferPnPRightVisionUnloadJob3(interlock := wire#w5, startCondition := wire#w8, parentReferenceDesignator := "Unit1.Em5.Config".em.referenceDesignator.combined, jobNumber := "U1EM5_JOB03", singleCycleJob := TRUE, hmiInterface := "Unit1.Em5.HmiInterface".transferPnPRight.jobs, jobs := "Unit1.Em5.ControlNodes".transferPnPRight.jobs, jobStatus => "Unit1.Em5.ControlNodes".transferPnPRight.selectJobStatus[3])
   END_RUNG
   RUNG wire#powerrail
      Contact( "Unit1.Em5.ControlNodes".em.status.initialized )
      Contact( #tempInterlockCond )
   END_RUNG wire#w5
   RUNG wire#powerrail
      Contact( #statUnitStatus.state.execute )
      I_Contact( #tempSpecialFunctionCheckbit )
      Contact( #tempPlaceCond )
      wire#w6
      I_Contact( #instTransferPnPRightVisionUnloadJob3.jobStatus.completed )
   END_RUNG wire#w8
   RUNG wire#powerrail
      Contact( #FALSE )
      wire#w7
      I_Contact( "Unit1.EmNodes".unitStatus.specialFunctions."Dry Run" )
      I_Contact( #statRoutingNok[1] )
   END_RUNG wire#w6
   RUNG wire#w7
      Contact( "Unit1.EmNodes".unitStatus.specialFunctions."Dry Run" )
   END_RUNG wire#w6
   // the same network as SCL:
   #tempInterlockCond := NOT #instTransferPnPRightVisionUnloadJob3.jobStatus.active AND NOT #instTransferPnPRightVisionLoadJob4.jobStatus.active AND NOT #instTransferPnPRightLaserMarkUnloadJob5.jobStatus.active AND NOT #instTransferPnPRightLaserMarkLoadJob6.jobStatus.active AND NOT #instTransferPnPRightWeightCheckUnloadJob9.jobStatus.active;
   #tempPickCond := "Unit1.EmNodes".emRelations.em08.cmStatus.HipotThicknessJRDetect.monitoring.processValue AND NOT "Unit1.Em5.ControlNodes".cmTransferPnPRightJRDetect.monitoring.processValue AND NOT "Unit1.EmNodes".emRelations.em09.sequence.vision.jobInterface.loadJob2.loadingDone AND "Unit1.EmNodes".emRelations.em08.sequence.hipotThickness.jobInterface.unloadJob4.unLoadingRequest;
   #instTransferPnPRightHipotThicknessLoadJob2(parentReferenceDesignator := "Unit1.Em5.Config".em.referenceDesignator.combined,   // "LAF_SelectJob"
                           jobNumber := "U1EM5_JOB02",
                           singleCycleJob := TRUE,
                           interlock := "Unit1.Em5.ControlNodes".em.status.initialized AND #tempInterlockCond,
                           startCondition := ((#statUnitStatus.state.execute AND NOT #tempSpecialFunctionCheckbit AND #tempPickCond) OR (false AND (#statRoutingOk[0] OR (#statRoutingNok[0] AND NOT "Unit1.EmNodes".emRelations.em10.sequence.laserMark.jobInterface.loadJob2.loadingDone) OR "Unit1.EmNodes".unitStatus.specialFunctions."Dry Run"))) AND NOT #instTransferPnPRightHipotThicknessLoadJob2.jobStatus.completed,
                           hmiInterface := "Unit1.Em5.HmiInterface".transferPnPRight.jobs,
                           jobs := "Unit1.Em5.ControlNodes".transferPnPRight.jobs,
                           jobStatus => "Unit1.Em5.ControlNodes".transferPnPRight.selectJobStatus[2]);
   #tempInterlockCond := NOT #instTransferPnPRightHipotThicknessLoadJob2.jobStatus.active AND NOT #instTransferPnPRightVisionLoadJob4.jobStatus.active AND NOT #instTransferPnPRightLaserMarkUnloadJob5.jobStatus.active AND NOT #instTransferPnPRightLaserMarkLoadJob6.jobStatus.active AND NOT #instTransferPnPRightWeightCheckUnloadJob9.jobStatus.active;
   #tempPlaceCond := "Unit1.Em5.ControlNodes".cmTransferPnPRightJRDetect.monitoring.processValue AND NOT "Unit1.EmNodes".emRelations.em09.cmStatus.VisionJRDetect.monitoring.processValue AND NOT "Unit1.EmNodes".emRelations.em09.sequence.vision.jobInterface.loadJob2.loadingDone AND "Unit1.EmNodes".emRelations.em09.sequence.vision.jobInterface.loadJob2.loadingRequest AND "Unit1.Em5.ControlNodes".transferPnPRight.jobInterface.hipotThicknessPICKJob2.workingDone;
   #instTransferPnPRightVisionUnloadJob3(parentReferenceDesignator := "Unit1.Em5.Config".em.referenceDesignator.combined,   // "LAF_SelectJob"
                           jobNumber := "U1EM5_JOB03",
                           singleCycleJob := TRUE,
                           interlock := "Unit1.Em5.ControlNodes".em.status.initialized AND #tempInterlockCond,
                           startCondition := ((#statUnitStatus.state.execute AND NOT #tempSpecialFunctionCheckbit AND #tempPlaceCond) OR (#FALSE AND ((NOT "Unit1.EmNodes".unitStatus.specialFunctions."Dry Run" AND NOT #statRoutingNok[1]) OR "Unit1.EmNodes".unitStatus.specialFunctions."Dry Run"))) AND NOT #instTransferPnPRightVisionUnloadJob3.jobStatus.completed,
                           hmiInterface := "Unit1.Em5.HmiInterface".transferPnPRight.jobs,
                           jobs := "Unit1.Em5.ControlNodes".transferPnPRight.jobs,
                           jobStatus => "Unit1.Em5.ControlNodes".transferPnPRight.selectJobStatus[3]);
END_REGION

REGION Network 47: Transfer P&P Right Job Interface [Hipot & Thickness Loading]
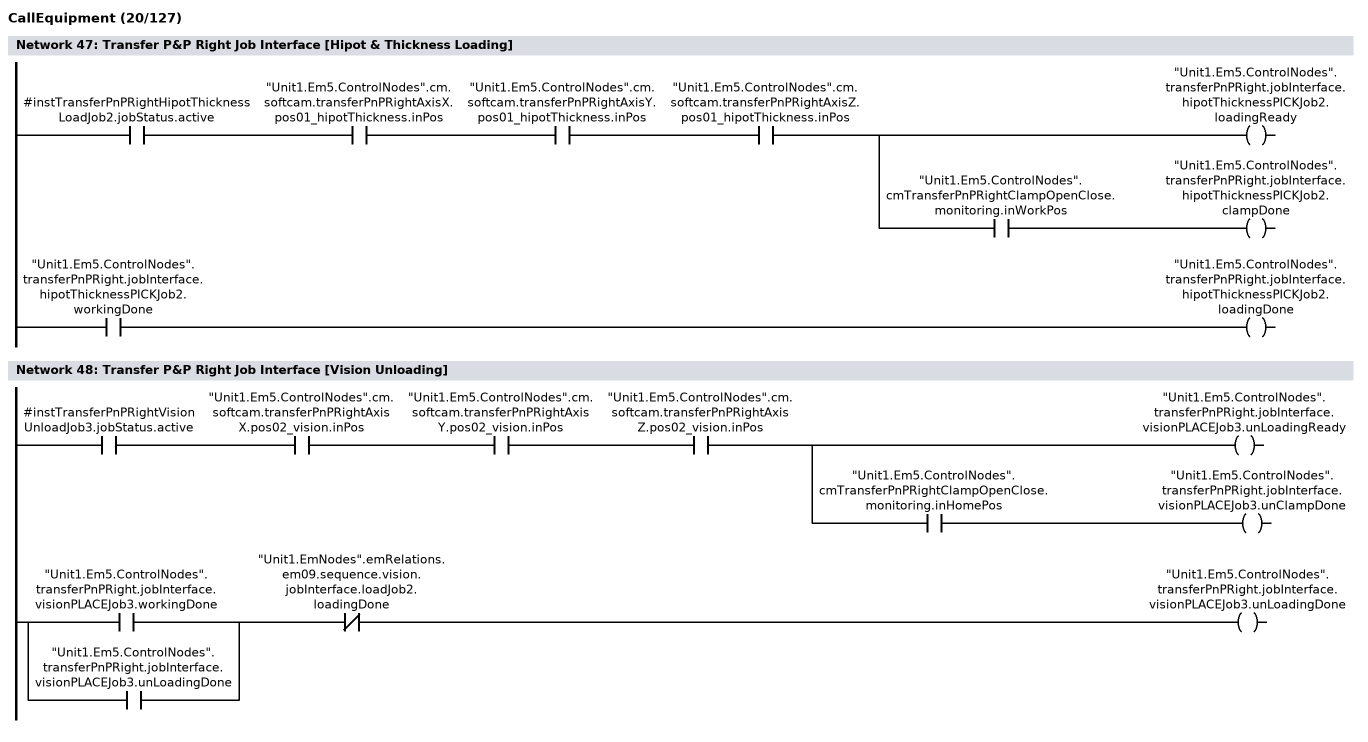
   RUNG wire#powerrail
      Contact( #instTransferPnPRightHipotThicknessLoadJob2.jobStatus.active )
      Contact( "Unit1.Em5.ControlNodes".cm.softcam.transferPnPRightAxisX.pos01_hipotThickness.inPos )
      Contact( "Unit1.Em5.ControlNodes".cm.softcam.transferPnPRightAxisY.pos01_hipotThickness.inPos )
      Contact( "Unit1.Em5.ControlNodes".cm.softcam.transferPnPRightAxisZ.pos01_hipotThickness.inPos )
      wire#w1
      Coil( "Unit1.Em5.ControlNodes".transferPnPRight.jobInterface.hipotThicknessPICKJob2.loadingReady )
   END_RUNG
   RUNG wire#w1
      Contact( "Unit1.Em5.ControlNodes".cmTransferPnPRightClampOpenClose.monitoring.inWorkPos )
      Coil( "Unit1.Em5.ControlNodes".transferPnPRight.jobInterface.hipotThicknessPICKJob2.clampDone )
   END_RUNG
   RUNG wire#powerrail
      Contact( "Unit1.Em5.ControlNodes".transferPnPRight.jobInterface.hipotThicknessPICKJob2.workingDone )
      Coil( "Unit1.Em5.ControlNodes".transferPnPRight.jobInterface.hipotThicknessPICKJob2.loadingDone )
   END_RUNG
   // the same network as SCL:
   "Unit1.Em5.ControlNodes".transferPnPRight.jobInterface.hipotThicknessPICKJob2.loadingReady := #instTransferPnPRightHipotThicknessLoadJob2.jobStatus.active AND "Unit1.Em5.ControlNodes".cm.softcam.transferPnPRightAxisX.pos01_hipotThickness.inPos AND "Unit1.Em5.ControlNodes".cm.softcam.transferPnPRightAxisY.pos01_hipotThickness.inPos AND "Unit1.Em5.ControlNodes".cm.softcam.transferPnPRightAxisZ.pos01_hipotThickness.inPos;
   "Unit1.Em5.ControlNodes".transferPnPRight.jobInterface.hipotThicknessPICKJob2.clampDone := "Unit1.Em5.ControlNodes".transferPnPRight.jobInterface.hipotThicknessPICKJob2.loadingReady AND "Unit1.Em5.ControlNodes".cmTransferPnPRightClampOpenClose.monitoring.inWorkPos;
   "Unit1.Em5.ControlNodes".transferPnPRight.jobInterface.hipotThicknessPICKJob2.loadingDone := "Unit1.Em5.ControlNodes".transferPnPRight.jobInterface.hipotThicknessPICKJob2.workingDone;
END_REGION

REGION Network 48: Transfer P&P Right Job Interface [Vision Unloading]
   RUNG wire#powerrail
      Contact( #instTransferPnPRightVisionUnloadJob3.jobStatus.active )
      Contact( "Unit1.Em5.ControlNodes".cm.softcam.transferPnPRightAxisX.pos02_vision.inPos )
      Contact( "Unit1.Em5.ControlNodes".cm.softcam.transferPnPRightAxisY.pos02_vision.inPos )
      Contact( "Unit1.Em5.ControlNodes".cm.softcam.transferPnPRightAxisZ.pos02_vision.inPos )
      wire#w1
      Coil( "Unit1.Em5.ControlNodes".transferPnPRight.jobInterface.visionPLACEJob3.unLoadingReady )
   END_RUNG
   RUNG wire#w1
      Contact( "Unit1.Em5.ControlNodes".cmTransferPnPRightClampOpenClose.monitoring.inHomePos )
      Coil( "Unit1.Em5.ControlNodes".transferPnPRight.jobInterface.visionPLACEJob3.unClampDone )
   END_RUNG
   RUNG wire#powerrail
      Contact( "Unit1.Em5.ControlNodes".transferPnPRight.jobInterface.visionPLACEJob3.workingDone )
      wire#w2
      I_Contact( "Unit1.EmNodes".emRelations.em09.sequence.vision.jobInterface.loadJob2.loadingDone )
      Coil( "Unit1.Em5.ControlNodes".transferPnPRight.jobInterface.visionPLACEJob3.unLoadingDone )
   END_RUNG
   RUNG wire#powerrail
      Contact( "Unit1.Em5.ControlNodes".transferPnPRight.jobInterface.visionPLACEJob3.unLoadingDone )
   END_RUNG wire#w2
   // the same network as SCL:
   "Unit1.Em5.ControlNodes".transferPnPRight.jobInterface.visionPLACEJob3.unLoadingReady := #instTransferPnPRightVisionUnloadJob3.jobStatus.active AND "Unit1.Em5.ControlNodes".cm.softcam.transferPnPRightAxisX.pos02_vision.inPos AND "Unit1.Em5.ControlNodes".cm.softcam.transferPnPRightAxisY.pos02_vision.inPos AND "Unit1.Em5.ControlNodes".cm.softcam.transferPnPRightAxisZ.pos02_vision.inPos;
   "Unit1.Em5.ControlNodes".transferPnPRight.jobInterface.visionPLACEJob3.unClampDone := "Unit1.Em5.ControlNodes".transferPnPRight.jobInterface.visionPLACEJob3.unLoadingReady AND "Unit1.Em5.ControlNodes".cmTransferPnPRightClampOpenClose.monitoring.inHomePos;
   "Unit1.Em5.ControlNodes".transferPnPRight.jobInterface.visionPLACEJob3.unLoadingDone := ("Unit1.Em5.ControlNodes".transferPnPRight.jobInterface.visionPLACEJob3.workingDone OR "Unit1.Em5.ControlNodes".transferPnPRight.jobInterface.visionPLACEJob3.unLoadingDone) AND NOT "Unit1.EmNodes".emRelations.em09.sequence.vision.jobInterface.loadJob2.loadingDone;
END_REGION

REGION Network 49: Transfer P&P Right Job Interface Working Done [Hipot & Thickness → Vision]
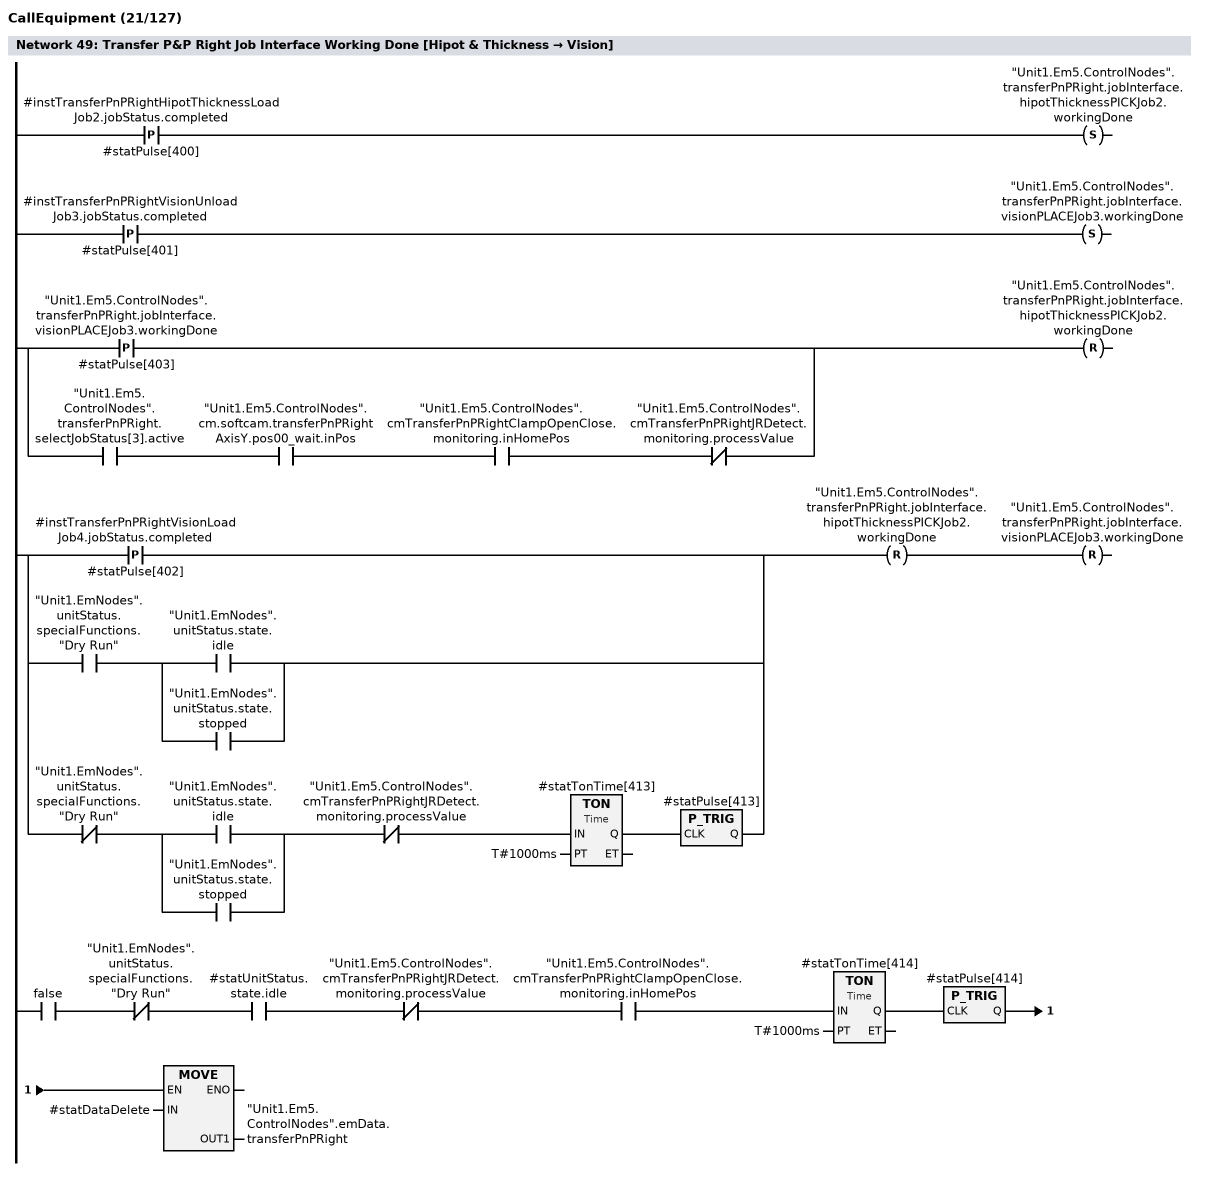
   RUNG wire#powerrail
      P_Contact(operand := #instTransferPnPRightHipotThicknessLoadJob2.jobStatus.completed, bit := #statPulse[400])
      S_Coil( "Unit1.Em5.ControlNodes".transferPnPRight.jobInterface.hipotThicknessPICKJob2.workingDone )
   END_RUNG
   RUNG wire#powerrail
      P_Contact(operand := #instTransferPnPRightVisionUnloadJob3.jobStatus.completed, bit := #statPulse[401])
      S_Coil( "Unit1.Em5.ControlNodes".transferPnPRight.jobInterface.visionPLACEJob3.workingDone )
   END_RUNG
   RUNG wire#powerrail
      P_Contact(operand := "Unit1.Em5.ControlNodes".transferPnPRight.jobInterface.visionPLACEJob3.workingDone, bit := #statPulse[403])
      wire#w1
      R_Coil( "Unit1.Em5.ControlNodes".transferPnPRight.jobInterface.hipotThicknessPICKJob2.workingDone )
   END_RUNG
   RUNG wire#powerrail
      Contact( "Unit1.Em5.ControlNodes".transferPnPRight.selectJobStatus[3].active )
      Contact( "Unit1.Em5.ControlNodes".cm.softcam.transferPnPRightAxisY.pos00_wait.inPos )
      Contact( "Unit1.Em5.ControlNodes".cmTransferPnPRightClampOpenClose.monitoring.inHomePos )
      I_Contact( "Unit1.Em5.ControlNodes".cmTransferPnPRightJRDetect.monitoring.processValue )
   END_RUNG wire#w1
   RUNG wire#powerrail
      P_Contact(operand := #instTransferPnPRightVisionLoadJob4.jobStatus.completed, bit := #statPulse[402])
      wire#w2
      R_Coil( "Unit1.Em5.ControlNodes".transferPnPRight.jobInterface.hipotThicknessPICKJob2.workingDone )
      R_Coil( "Unit1.Em5.ControlNodes".transferPnPRight.jobInterface.visionPLACEJob3.workingDone )
   END_RUNG
   RUNG wire#powerrail
      Contact( "Unit1.EmNodes".unitStatus.specialFunctions."Dry Run" )
      wire#w3
      Contact( "Unit1.EmNodes".unitStatus.state.idle )
   END_RUNG wire#w2
   RUNG wire#w3
      Contact( "Unit1.EmNodes".unitStatus.state.stopped )
   END_RUNG wire#w2
   RUNG wire#powerrail
      I_Contact( "Unit1.EmNodes".unitStatus.specialFunctions."Dry Run" )
      wire#w4
      Contact( "Unit1.EmNodes".unitStatus.state.idle )
      wire#w5
      I_Contact( "Unit1.Em5.ControlNodes".cmTransferPnPRightJRDetect.monitoring.processValue )
      { S7_Templates := "time_type := Time" } #statTonTime[413].TON(pt := T#1000ms, et =>)
      P_Trig( #statPulse[413] )
   END_RUNG wire#w2
   RUNG wire#w4
      Contact( "Unit1.EmNodes".unitStatus.state.stopped )
   END_RUNG wire#w5
   RUNG wire#powerrail
      Contact( false )
      I_Contact( "Unit1.EmNodes".unitStatus.specialFunctions."Dry Run" )
      Contact( #statUnitStatus.state.idle )
      I_Contact( "Unit1.Em5.ControlNodes".cmTransferPnPRightJRDetect.monitoring.processValue )
      Contact( "Unit1.Em5.ControlNodes".cmTransferPnPRightClampOpenClose.monitoring.inHomePos )
      { S7_Templates := "time_type := Time" } #statTonTime[414].TON(pt := T#1000ms, et =>)
      P_Trig( #statPulse[414] )
      Move(in := #statDataDelete, out1 => "Unit1.Em5.ControlNodes".emData.transferPnPRight)
   END_RUNG
   // the same network as SCL:
   #_w1 := #instTransferPnPRightHipotThicknessLoadJob2.jobStatus.completed AND NOT #statPulse[400];   // rising edge of #instTransferPnPRightHipotThicknessLoadJob2.jobStatus.completed
   #statPulse[400] := #instTransferPnPRightHipotThicknessLoadJob2.jobStatus.completed;
   IF #_w1 THEN
       "Unit1.Em5.ControlNodes".transferPnPRight.jobInterface.hipotThicknessPICKJob2.workingDone := TRUE;
   END_IF;
   #_w2 := #instTransferPnPRightVisionUnloadJob3.jobStatus.completed AND NOT #statPulse[401];   // rising edge of #instTransferPnPRightVisionUnloadJob3.jobStatus.completed
   #statPulse[401] := #instTransferPnPRightVisionUnloadJob3.jobStatus.completed;
   IF #_w2 THEN
       "Unit1.Em5.ControlNodes".transferPnPRight.jobInterface.visionPLACEJob3.workingDone := TRUE;
   END_IF;
   #_w3 := "Unit1.Em5.ControlNodes".transferPnPRight.jobInterface.visionPLACEJob3.workingDone AND NOT #statPulse[403];   // rising edge of "Unit1.Em5.ControlNodes".transferPnPRight.jobInterface.visionPLACEJob3.workingDone
   #statPulse[403] := "Unit1.Em5.ControlNodes".transferPnPRight.jobInterface.visionPLACEJob3.workingDone;
   IF #_w3 OR ("Unit1.Em5.ControlNodes".transferPnPRight.selectJobStatus[3].active AND "Unit1.Em5.ControlNodes".cm.softcam.transferPnPRightAxisY.pos00_wait.inPos AND "Unit1.Em5.ControlNodes".cmTransferPnPRightClampOpenClose.monitoring.inHomePos AND NOT "Unit1.Em5.ControlNodes".cmTransferPnPRightJRDetect.monitoring.processValue) THEN
       "Unit1.Em5.ControlNodes".transferPnPRight.jobInterface.hipotThicknessPICKJob2.workingDone := FALSE;
   END_IF;
   #_w4 := #instTransferPnPRightVisionLoadJob4.jobStatus.completed AND NOT #statPulse[402];   // rising edge of #instTransferPnPRightVisionLoadJob4.jobStatus.completed
   #statPulse[402] := #instTransferPnPRightVisionLoadJob4.jobStatus.completed;
   #statTonTime[413].TON(IN := NOT "Unit1.EmNodes".unitStatus.specialFunctions."Dry Run" AND ("Unit1.EmNodes".unitStatus.state.idle OR "Unit1.EmNodes".unitStatus.state.stopped) AND NOT "Unit1.Em5.ControlNodes".cmTransferPnPRightJRDetect.monitoring.processValue,
                         PT := T#1000ms);
   #_w5 := #statTonTime[413].Q AND NOT #statPulse[413];   // rising edge
   #statPulse[413] := #statTonTime[413].Q;
   IF #_w4 OR ("Unit1.EmNodes".unitStatus.specialFunctions."Dry Run" AND ("Unit1.EmNodes".unitStatus.state.idle OR "Unit1.EmNodes".unitStatus.state.stopped)) OR #_w5 THEN
       "Unit1.Em5.ControlNodes".transferPnPRight.jobInterface.hipotThicknessPICKJob2.workingDone := FALSE;
       "Unit1.Em5.ControlNodes".transferPnPRight.jobInterface.visionPLACEJob3.workingDone := FALSE;
   END_IF;
   #statTonTime[414].TON(IN := false AND NOT "Unit1.EmNodes".unitStatus.specialFunctions."Dry Run" AND #statUnitStatus.state.idle AND NOT "Unit1.Em5.ControlNodes".cmTransferPnPRightJRDetect.monitoring.processValue AND "Unit1.Em5.ControlNodes".cmTransferPnPRightClampOpenClose.monitoring.inHomePos,
                         PT := T#1000ms);
   #_w6 := #statTonTime[414].Q AND NOT #statPulse[414];   // rising edge
   #statPulse[414] := #statTonTime[414].Q;
   IF #_w6 THEN "Unit1.Em5.ControlNodes".emData.transferPnPRight := #statDataDelete; END_IF;
END_REGION

REGION Network 51: [Job] Transfer P&P Right Select Job
   // Configure here when the jobs of the sequence should be started. More jobs could be added.
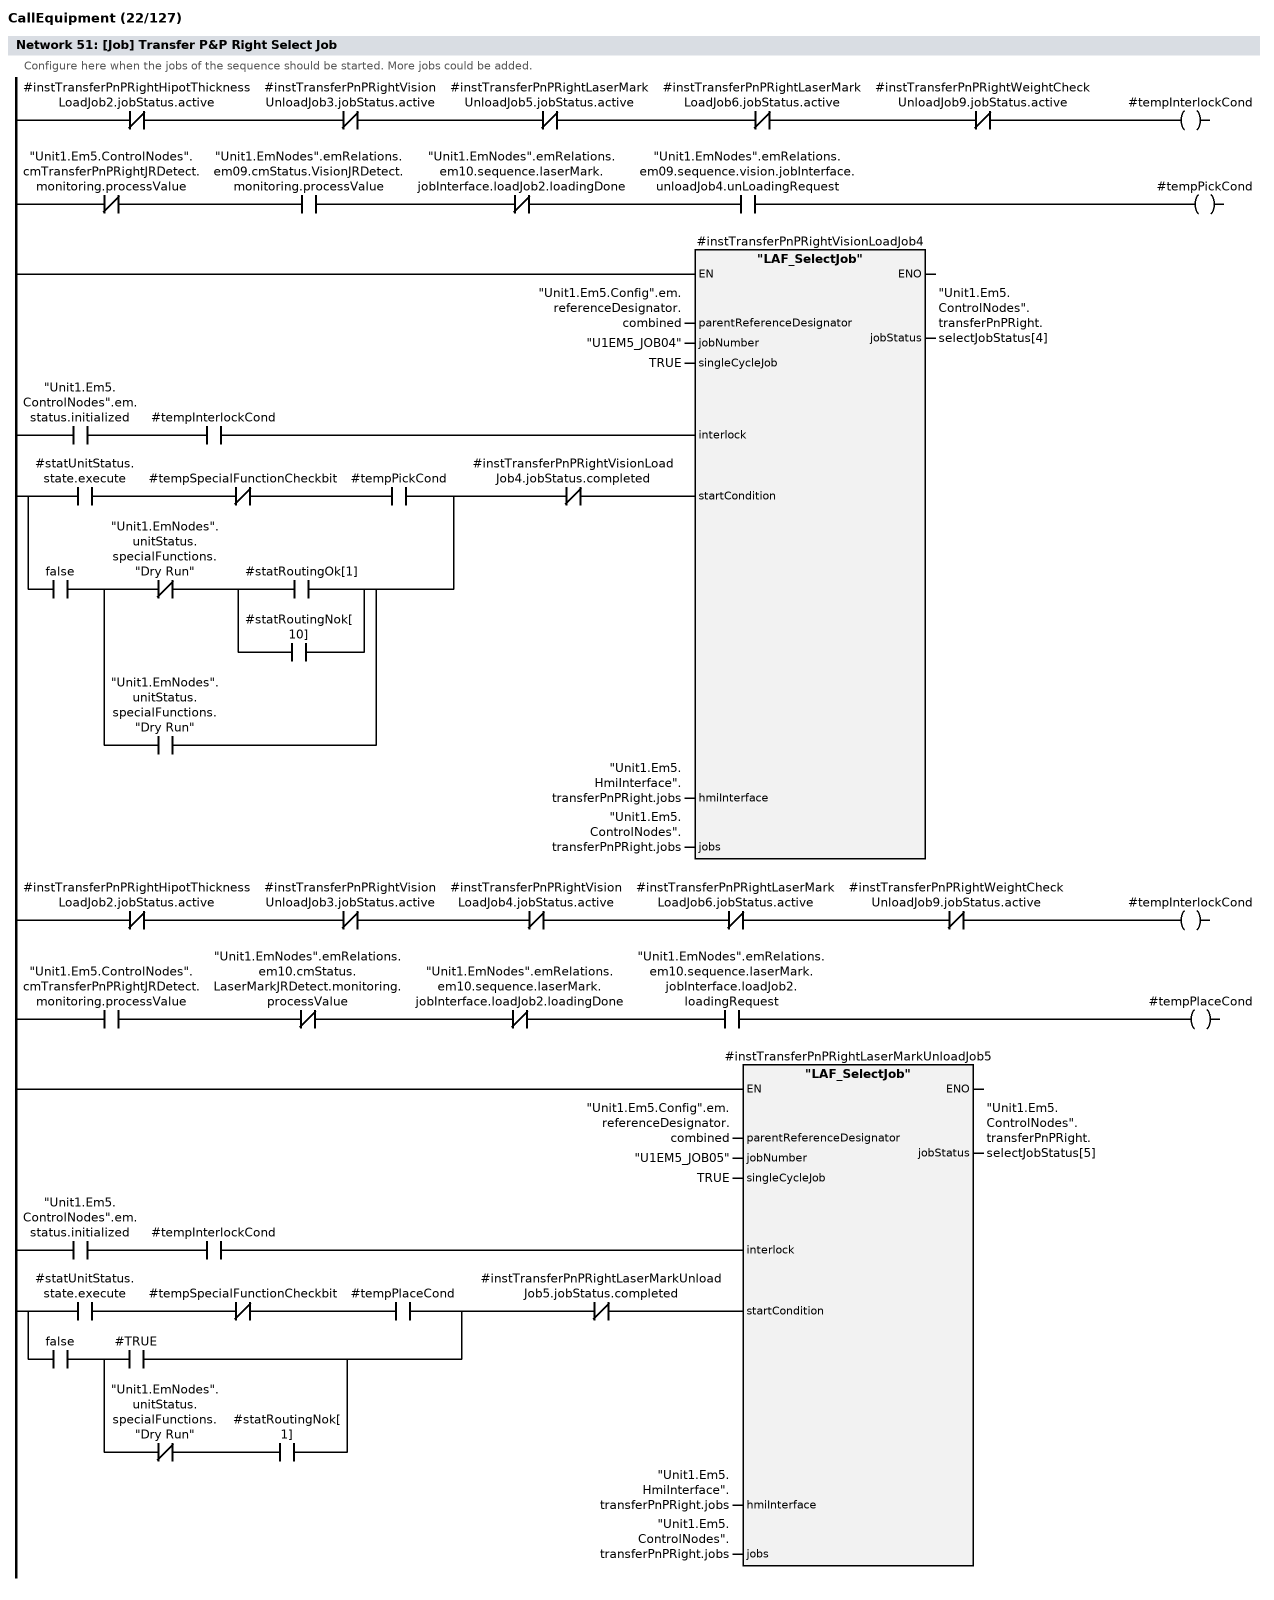
   RUNG wire#powerrail
      I_Contact( #instTransferPnPRightHipotThicknessLoadJob2.jobStatus.active )
      I_Contact( #instTransferPnPRightVisionUnloadJob3.jobStatus.active )
      I_Contact( #instTransferPnPRightLaserMarkUnloadJob5.jobStatus.active )
      I_Contact( #instTransferPnPRightLaserMarkLoadJob6.jobStatus.active )
      I_Contact( #instTransferPnPRightWeightCheckUnloadJob9.jobStatus.active )
      Coil( #tempInterlockCond )
   END_RUNG
   RUNG wire#powerrail
      I_Contact( "Unit1.Em5.ControlNodes".cmTransferPnPRightJRDetect.monitoring.processValue )
      Contact( "Unit1.EmNodes".emRelations.em09.cmStatus.VisionJRDetect.monitoring.processValue )
      I_Contact( "Unit1.EmNodes".emRelations.em10.sequence.laserMark.jobInterface.loadJob2.loadingDone )
      Contact( "Unit1.EmNodes".emRelations.em09.sequence.vision.jobInterface.unloadJob4.unLoadingRequest )
      Coil( #tempPickCond )
   END_RUNG
   RUNG wire#powerrail
      #instTransferPnPRightVisionLoadJob4(interlock := wire#w1, startCondition := wire#w5, parentReferenceDesignator := "Unit1.Em5.Config".em.referenceDesignator.combined, jobNumber := "U1EM5_JOB04", singleCycleJob := TRUE, hmiInterface := "Unit1.Em5.HmiInterface".transferPnPRight.jobs, jobs := "Unit1.Em5.ControlNodes".transferPnPRight.jobs, jobStatus => "Unit1.Em5.ControlNodes".transferPnPRight.selectJobStatus[4])
   END_RUNG
   RUNG wire#powerrail
      Contact( "Unit1.Em5.ControlNodes".em.status.initialized )
      Contact( #tempInterlockCond )
   END_RUNG wire#w1
   RUNG wire#powerrail
      Contact( #statUnitStatus.state.execute )
      I_Contact( #tempSpecialFunctionCheckbit )
      Contact( #tempPickCond )
      wire#w2
      I_Contact( #instTransferPnPRightVisionLoadJob4.jobStatus.completed )
   END_RUNG wire#w5
   RUNG wire#powerrail
      Contact( false )
      wire#w3
      I_Contact( "Unit1.EmNodes".unitStatus.specialFunctions."Dry Run" )
      wire#w4
      Contact( #statRoutingOk[1] )
   END_RUNG wire#w2
   RUNG wire#w4
      Contact( #statRoutingNok[10] )
   END_RUNG wire#w2
   RUNG wire#w3
      Contact( "Unit1.EmNodes".unitStatus.specialFunctions."Dry Run" )
   END_RUNG wire#w2
   RUNG wire#powerrail
      I_Contact( #instTransferPnPRightHipotThicknessLoadJob2.jobStatus.active )
      I_Contact( #instTransferPnPRightVisionUnloadJob3.jobStatus.active )
      I_Contact( #instTransferPnPRightVisionLoadJob4.jobStatus.active )
      I_Contact( #instTransferPnPRightLaserMarkLoadJob6.jobStatus.active )
      I_Contact( #instTransferPnPRightWeightCheckUnloadJob9.jobStatus.active )
      Coil( #tempInterlockCond )
   END_RUNG
   RUNG wire#powerrail
      Contact( "Unit1.Em5.ControlNodes".cmTransferPnPRightJRDetect.monitoring.processValue )
      I_Contact( "Unit1.EmNodes".emRelations.em10.cmStatus.LaserMarkJRDetect.monitoring.processValue )
      I_Contact( "Unit1.EmNodes".emRelations.em10.sequence.laserMark.jobInterface.loadJob2.loadingDone )
      Contact( "Unit1.EmNodes".emRelations.em10.sequence.laserMark.jobInterface.loadJob2.loadingRequest )
      Coil( #tempPlaceCond )
   END_RUNG
   RUNG wire#powerrail
      #instTransferPnPRightLaserMarkUnloadJob5(interlock := wire#w6, startCondition := wire#w9, parentReferenceDesignator := "Unit1.Em5.Config".em.referenceDesignator.combined, jobNumber := "U1EM5_JOB05", singleCycleJob := TRUE, hmiInterface := "Unit1.Em5.HmiInterface".transferPnPRight.jobs, jobs := "Unit1.Em5.ControlNodes".transferPnPRight.jobs, jobStatus => "Unit1.Em5.ControlNodes".transferPnPRight.selectJobStatus[5])
   END_RUNG
   RUNG wire#powerrail
      Contact( "Unit1.Em5.ControlNodes".em.status.initialized )
      Contact( #tempInterlockCond )
   END_RUNG wire#w6
   RUNG wire#powerrail
      Contact( #statUnitStatus.state.execute )
      I_Contact( #tempSpecialFunctionCheckbit )
      Contact( #tempPlaceCond )
      wire#w7
      I_Contact( #instTransferPnPRightLaserMarkUnloadJob5.jobStatus.completed )
   END_RUNG wire#w9
   RUNG wire#powerrail
      Contact( false )
      wire#w8
      Contact( #TRUE )
   END_RUNG wire#w7
   RUNG wire#w8
      I_Contact( "Unit1.EmNodes".unitStatus.specialFunctions."Dry Run" )
      Contact( #statRoutingNok[1] )
   END_RUNG wire#w7
   // the same network as SCL:
   #tempInterlockCond := NOT #instTransferPnPRightHipotThicknessLoadJob2.jobStatus.active AND NOT #instTransferPnPRightVisionUnloadJob3.jobStatus.active AND NOT #instTransferPnPRightLaserMarkUnloadJob5.jobStatus.active AND NOT #instTransferPnPRightLaserMarkLoadJob6.jobStatus.active AND NOT #instTransferPnPRightWeightCheckUnloadJob9.jobStatus.active;
   #tempPickCond := NOT "Unit1.Em5.ControlNodes".cmTransferPnPRightJRDetect.monitoring.processValue AND "Unit1.EmNodes".emRelations.em09.cmStatus.VisionJRDetect.monitoring.processValue AND NOT "Unit1.EmNodes".emRelations.em10.sequence.laserMark.jobInterface.loadJob2.loadingDone AND "Unit1.EmNodes".emRelations.em09.sequence.vision.jobInterface.unloadJob4.unLoadingRequest;
   #instTransferPnPRightVisionLoadJob4(parentReferenceDesignator := "Unit1.Em5.Config".em.referenceDesignator.combined,   // "LAF_SelectJob"
                           jobNumber := "U1EM5_JOB04",
                           singleCycleJob := TRUE,
                           interlock := "Unit1.Em5.ControlNodes".em.status.initialized AND #tempInterlockCond,
                           startCondition := ((#statUnitStatus.state.execute AND NOT #tempSpecialFunctionCheckbit AND #tempPickCond) OR (false AND ((NOT "Unit1.EmNodes".unitStatus.specialFunctions."Dry Run" AND (#statRoutingOk[1] OR #statRoutingNok[10])) OR "Unit1.EmNodes".unitStatus.specialFunctions."Dry Run"))) AND NOT #instTransferPnPRightVisionLoadJob4.jobStatus.completed,
                           hmiInterface := "Unit1.Em5.HmiInterface".transferPnPRight.jobs,
                           jobs := "Unit1.Em5.ControlNodes".transferPnPRight.jobs,
                           jobStatus => "Unit1.Em5.ControlNodes".transferPnPRight.selectJobStatus[4]);
   #tempInterlockCond := NOT #instTransferPnPRightHipotThicknessLoadJob2.jobStatus.active AND NOT #instTransferPnPRightVisionUnloadJob3.jobStatus.active AND NOT #instTransferPnPRightVisionLoadJob4.jobStatus.active AND NOT #instTransferPnPRightLaserMarkLoadJob6.jobStatus.active AND NOT #instTransferPnPRightWeightCheckUnloadJob9.jobStatus.active;
   #tempPlaceCond := "Unit1.Em5.ControlNodes".cmTransferPnPRightJRDetect.monitoring.processValue AND NOT "Unit1.EmNodes".emRelations.em10.cmStatus.LaserMarkJRDetect.monitoring.processValue AND NOT "Unit1.EmNodes".emRelations.em10.sequence.laserMark.jobInterface.loadJob2.loadingDone AND "Unit1.EmNodes".emRelations.em10.sequence.laserMark.jobInterface.loadJob2.loadingRequest;
   #instTransferPnPRightLaserMarkUnloadJob5(parentReferenceDesignator := "Unit1.Em5.Config".em.referenceDesignator.combined,   // "LAF_SelectJob"
                           jobNumber := "U1EM5_JOB05",
                           singleCycleJob := TRUE,
                           interlock := "Unit1.Em5.ControlNodes".em.status.initialized AND #tempInterlockCond,
                           startCondition := ((#statUnitStatus.state.execute AND NOT #tempSpecialFunctionCheckbit AND #tempPlaceCond) OR (false AND (#TRUE OR (NOT "Unit1.EmNodes".unitStatus.specialFunctions."Dry Run" AND #statRoutingNok[1])))) AND NOT #instTransferPnPRightLaserMarkUnloadJob5.jobStatus.completed,
                           hmiInterface := "Unit1.Em5.HmiInterface".transferPnPRight.jobs,
                           jobs := "Unit1.Em5.ControlNodes".transferPnPRight.jobs,
                           jobStatus => "Unit1.Em5.ControlNodes".transferPnPRight.selectJobStatus[5]);
END_REGION

REGION Network 52: Transfer P&P Right Job Interface [Vision Loading]
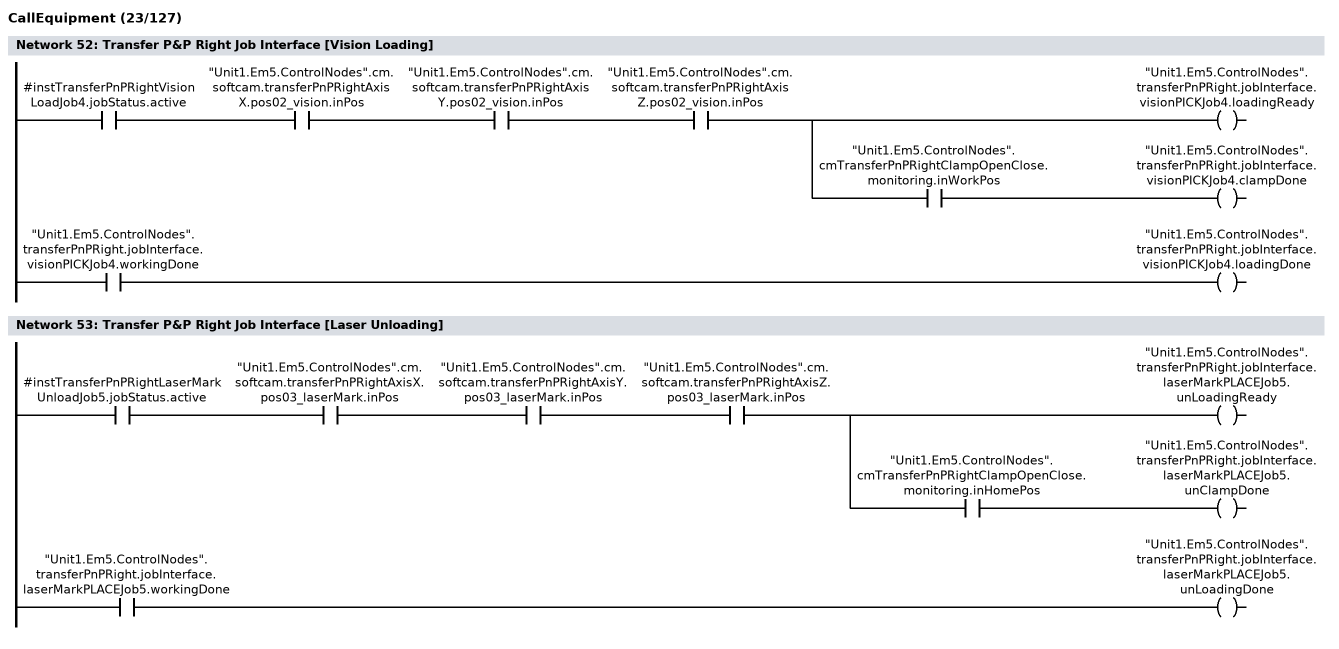
   RUNG wire#powerrail
      Contact( #instTransferPnPRightVisionLoadJob4.jobStatus.active )
      Contact( "Unit1.Em5.ControlNodes".cm.softcam.transferPnPRightAxisX.pos02_vision.inPos )
      Contact( "Unit1.Em5.ControlNodes".cm.softcam.transferPnPRightAxisY.pos02_vision.inPos )
      Contact( "Unit1.Em5.ControlNodes".cm.softcam.transferPnPRightAxisZ.pos02_vision.inPos )
      wire#w1
      Coil( "Unit1.Em5.ControlNodes".transferPnPRight.jobInterface.visionPICKJob4.loadingReady )
   END_RUNG
   RUNG wire#w1
      Contact( "Unit1.Em5.ControlNodes".cmTransferPnPRightClampOpenClose.monitoring.inWorkPos )
      Coil( "Unit1.Em5.ControlNodes".transferPnPRight.jobInterface.visionPICKJob4.clampDone )
   END_RUNG
   RUNG wire#powerrail
      Contact( "Unit1.Em5.ControlNodes".transferPnPRight.jobInterface.visionPICKJob4.workingDone )
      Coil( "Unit1.Em5.ControlNodes".transferPnPRight.jobInterface.visionPICKJob4.loadingDone )
   END_RUNG
   // the same network as SCL:
   "Unit1.Em5.ControlNodes".transferPnPRight.jobInterface.visionPICKJob4.loadingReady := #instTransferPnPRightVisionLoadJob4.jobStatus.active AND "Unit1.Em5.ControlNodes".cm.softcam.transferPnPRightAxisX.pos02_vision.inPos AND "Unit1.Em5.ControlNodes".cm.softcam.transferPnPRightAxisY.pos02_vision.inPos AND "Unit1.Em5.ControlNodes".cm.softcam.transferPnPRightAxisZ.pos02_vision.inPos;
   "Unit1.Em5.ControlNodes".transferPnPRight.jobInterface.visionPICKJob4.clampDone := "Unit1.Em5.ControlNodes".transferPnPRight.jobInterface.visionPICKJob4.loadingReady AND "Unit1.Em5.ControlNodes".cmTransferPnPRightClampOpenClose.monitoring.inWorkPos;
   "Unit1.Em5.ControlNodes".transferPnPRight.jobInterface.visionPICKJob4.loadingDone := "Unit1.Em5.ControlNodes".transferPnPRight.jobInterface.visionPICKJob4.workingDone;
END_REGION

REGION Network 53: Transfer P&P Right Job Interface [Laser Unloading]
   RUNG wire#powerrail
      Contact( #instTransferPnPRightLaserMarkUnloadJob5.jobStatus.active )
      Contact( "Unit1.Em5.ControlNodes".cm.softcam.transferPnPRightAxisX.pos03_laserMark.inPos )
      Contact( "Unit1.Em5.ControlNodes".cm.softcam.transferPnPRightAxisY.pos03_laserMark.inPos )
      Contact( "Unit1.Em5.ControlNodes".cm.softcam.transferPnPRightAxisZ.pos03_laserMark.inPos )
      wire#w1
      Coil( "Unit1.Em5.ControlNodes".transferPnPRight.jobInterface.laserMarkPLACEJob5.unLoadingReady )
   END_RUNG
   RUNG wire#w1
      Contact( "Unit1.Em5.ControlNodes".cmTransferPnPRightClampOpenClose.monitoring.inHomePos )
      Coil( "Unit1.Em5.ControlNodes".transferPnPRight.jobInterface.laserMarkPLACEJob5.unClampDone )
   END_RUNG
   RUNG wire#powerrail
      Contact( "Unit1.Em5.ControlNodes".transferPnPRight.jobInterface.laserMarkPLACEJob5.workingDone )
      Coil( "Unit1.Em5.ControlNodes".transferPnPRight.jobInterface.laserMarkPLACEJob5.unLoadingDone )
   END_RUNG
   // the same network as SCL:
   "Unit1.Em5.ControlNodes".transferPnPRight.jobInterface.laserMarkPLACEJob5.unLoadingReady := #instTransferPnPRightLaserMarkUnloadJob5.jobStatus.active AND "Unit1.Em5.ControlNodes".cm.softcam.transferPnPRightAxisX.pos03_laserMark.inPos AND "Unit1.Em5.ControlNodes".cm.softcam.transferPnPRightAxisY.pos03_laserMark.inPos AND "Unit1.Em5.ControlNodes".cm.softcam.transferPnPRightAxisZ.pos03_laserMark.inPos;
   "Unit1.Em5.ControlNodes".transferPnPRight.jobInterface.laserMarkPLACEJob5.unClampDone := "Unit1.Em5.ControlNodes".transferPnPRight.jobInterface.laserMarkPLACEJob5.unLoadingReady AND "Unit1.Em5.ControlNodes".cmTransferPnPRightClampOpenClose.monitoring.inHomePos;
   "Unit1.Em5.ControlNodes".transferPnPRight.jobInterface.laserMarkPLACEJob5.unLoadingDone := "Unit1.Em5.ControlNodes".transferPnPRight.jobInterface.laserMarkPLACEJob5.workingDone;
END_REGION

REGION Network 54: Transfer P&P Right Job Interface Working Done [Vision → Laser Mark]
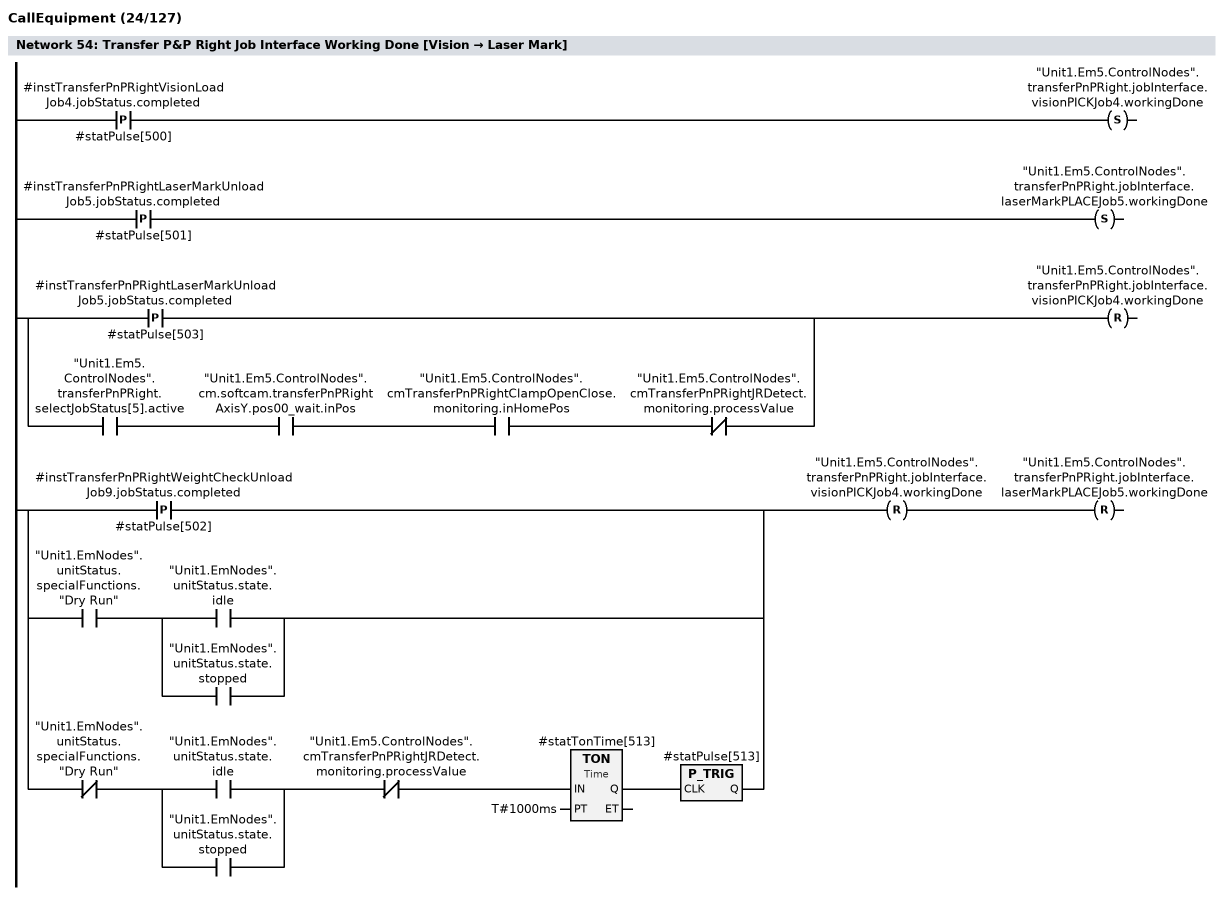
   RUNG wire#powerrail
      P_Contact(operand := #instTransferPnPRightVisionLoadJob4.jobStatus.completed, bit := #statPulse[500])
      S_Coil( "Unit1.Em5.ControlNodes".transferPnPRight.jobInterface.visionPICKJob4.workingDone )
   END_RUNG
   RUNG wire#powerrail
      P_Contact(operand := #instTransferPnPRightLaserMarkUnloadJob5.jobStatus.completed, bit := #statPulse[501])
      S_Coil( "Unit1.Em5.ControlNodes".transferPnPRight.jobInterface.laserMarkPLACEJob5.workingDone )
   END_RUNG
   RUNG wire#powerrail
      P_Contact(operand := #instTransferPnPRightLaserMarkUnloadJob5.jobStatus.completed, bit := #statPulse[503])
      wire#w1
      R_Coil( "Unit1.Em5.ControlNodes".transferPnPRight.jobInterface.visionPICKJob4.workingDone )
   END_RUNG
   RUNG wire#powerrail
      Contact( "Unit1.Em5.ControlNodes".transferPnPRight.selectJobStatus[5].active )
      Contact( "Unit1.Em5.ControlNodes".cm.softcam.transferPnPRightAxisY.pos00_wait.inPos )
      Contact( "Unit1.Em5.ControlNodes".cmTransferPnPRightClampOpenClose.monitoring.inHomePos )
      I_Contact( "Unit1.Em5.ControlNodes".cmTransferPnPRightJRDetect.monitoring.processValue )
   END_RUNG wire#w1
   RUNG wire#powerrail
      P_Contact(operand := #instTransferPnPRightWeightCheckUnloadJob9.jobStatus.completed, bit := #statPulse[502])
      wire#w2
      R_Coil( "Unit1.Em5.ControlNodes".transferPnPRight.jobInterface.visionPICKJob4.workingDone )
      R_Coil( "Unit1.Em5.ControlNodes".transferPnPRight.jobInterface.laserMarkPLACEJob5.workingDone )
   END_RUNG
   RUNG wire#powerrail
      Contact( "Unit1.EmNodes".unitStatus.specialFunctions."Dry Run" )
      wire#w3
      Contact( "Unit1.EmNodes".unitStatus.state.idle )
   END_RUNG wire#w2
   RUNG wire#w3
      Contact( "Unit1.EmNodes".unitStatus.state.stopped )
   END_RUNG wire#w2
   RUNG wire#powerrail
      I_Contact( "Unit1.EmNodes".unitStatus.specialFunctions."Dry Run" )
      wire#w4
      Contact( "Unit1.EmNodes".unitStatus.state.idle )
      wire#w5
      I_Contact( "Unit1.Em5.ControlNodes".cmTransferPnPRightJRDetect.monitoring.processValue )
      { S7_Templates := "time_type := Time" } #statTonTime[513].TON(pt := T#1000ms, et =>)
      P_Trig( #statPulse[513] )
   END_RUNG wire#w2
   RUNG wire#w4
      Contact( "Unit1.EmNodes".unitStatus.state.stopped )
   END_RUNG wire#w5
   // the same network as SCL:
   #_w1 := #instTransferPnPRightVisionLoadJob4.jobStatus.completed AND NOT #statPulse[500];   // rising edge of #instTransferPnPRightVisionLoadJob4.jobStatus.completed
   #statPulse[500] := #instTransferPnPRightVisionLoadJob4.jobStatus.completed;
   IF #_w1 THEN
       "Unit1.Em5.ControlNodes".transferPnPRight.jobInterface.visionPICKJob4.workingDone := TRUE;
   END_IF;
   #_w2 := #instTransferPnPRightLaserMarkUnloadJob5.jobStatus.completed AND NOT #statPulse[501];   // rising edge of #instTransferPnPRightLaserMarkUnloadJob5.jobStatus.completed
   #statPulse[501] := #instTransferPnPRightLaserMarkUnloadJob5.jobStatus.completed;
   IF #_w2 THEN
       "Unit1.Em5.ControlNodes".transferPnPRight.jobInterface.laserMarkPLACEJob5.workingDone := TRUE;
   END_IF;
   #_w3 := #instTransferPnPRightLaserMarkUnloadJob5.jobStatus.completed AND NOT #statPulse[503];   // rising edge of #instTransferPnPRightLaserMarkUnloadJob5.jobStatus.completed
   #statPulse[503] := #instTransferPnPRightLaserMarkUnloadJob5.jobStatus.completed;
   IF #_w3 OR ("Unit1.Em5.ControlNodes".transferPnPRight.selectJobStatus[5].active AND "Unit1.Em5.ControlNodes".cm.softcam.transferPnPRightAxisY.pos00_wait.inPos AND "Unit1.Em5.ControlNodes".cmTransferPnPRightClampOpenClose.monitoring.inHomePos AND NOT "Unit1.Em5.ControlNodes".cmTransferPnPRightJRDetect.monitoring.processValue) THEN
       "Unit1.Em5.ControlNodes".transferPnPRight.jobInterface.visionPICKJob4.workingDone := FALSE;
   END_IF;
   #_w4 := #instTransferPnPRightWeightCheckUnloadJob9.jobStatus.completed AND NOT #statPulse[502];   // rising edge of #instTransferPnPRightWeightCheckUnloadJob9.jobStatus.completed
   #statPulse[502] := #instTransferPnPRightWeightCheckUnloadJob9.jobStatus.completed;
   #statTonTime[513].TON(IN := NOT "Unit1.EmNodes".unitStatus.specialFunctions."Dry Run" AND ("Unit1.EmNodes".unitStatus.state.idle OR "Unit1.EmNodes".unitStatus.state.stopped) AND NOT "Unit1.Em5.ControlNodes".cmTransferPnPRightJRDetect.monitoring.processValue,
                         PT := T#1000ms);
   #_w5 := #statTonTime[513].Q AND NOT #statPulse[513];   // rising edge
   #statPulse[513] := #statTonTime[513].Q;
   IF #_w4 OR ("Unit1.EmNodes".unitStatus.specialFunctions."Dry Run" AND ("Unit1.EmNodes".unitStatus.state.idle OR "Unit1.EmNodes".unitStatus.state.stopped)) OR #_w5 THEN
       "Unit1.Em5.ControlNodes".transferPnPRight.jobInterface.visionPICKJob4.workingDone := FALSE;
       "Unit1.Em5.ControlNodes".transferPnPRight.jobInterface.laserMarkPLACEJob5.workingDone := FALSE;
   END_IF;
END_REGION

REGION Network 56: [Job] Transfer P&P Right Select Job
   // Configure here when the jobs of the sequence should be started. More jobs could be added.
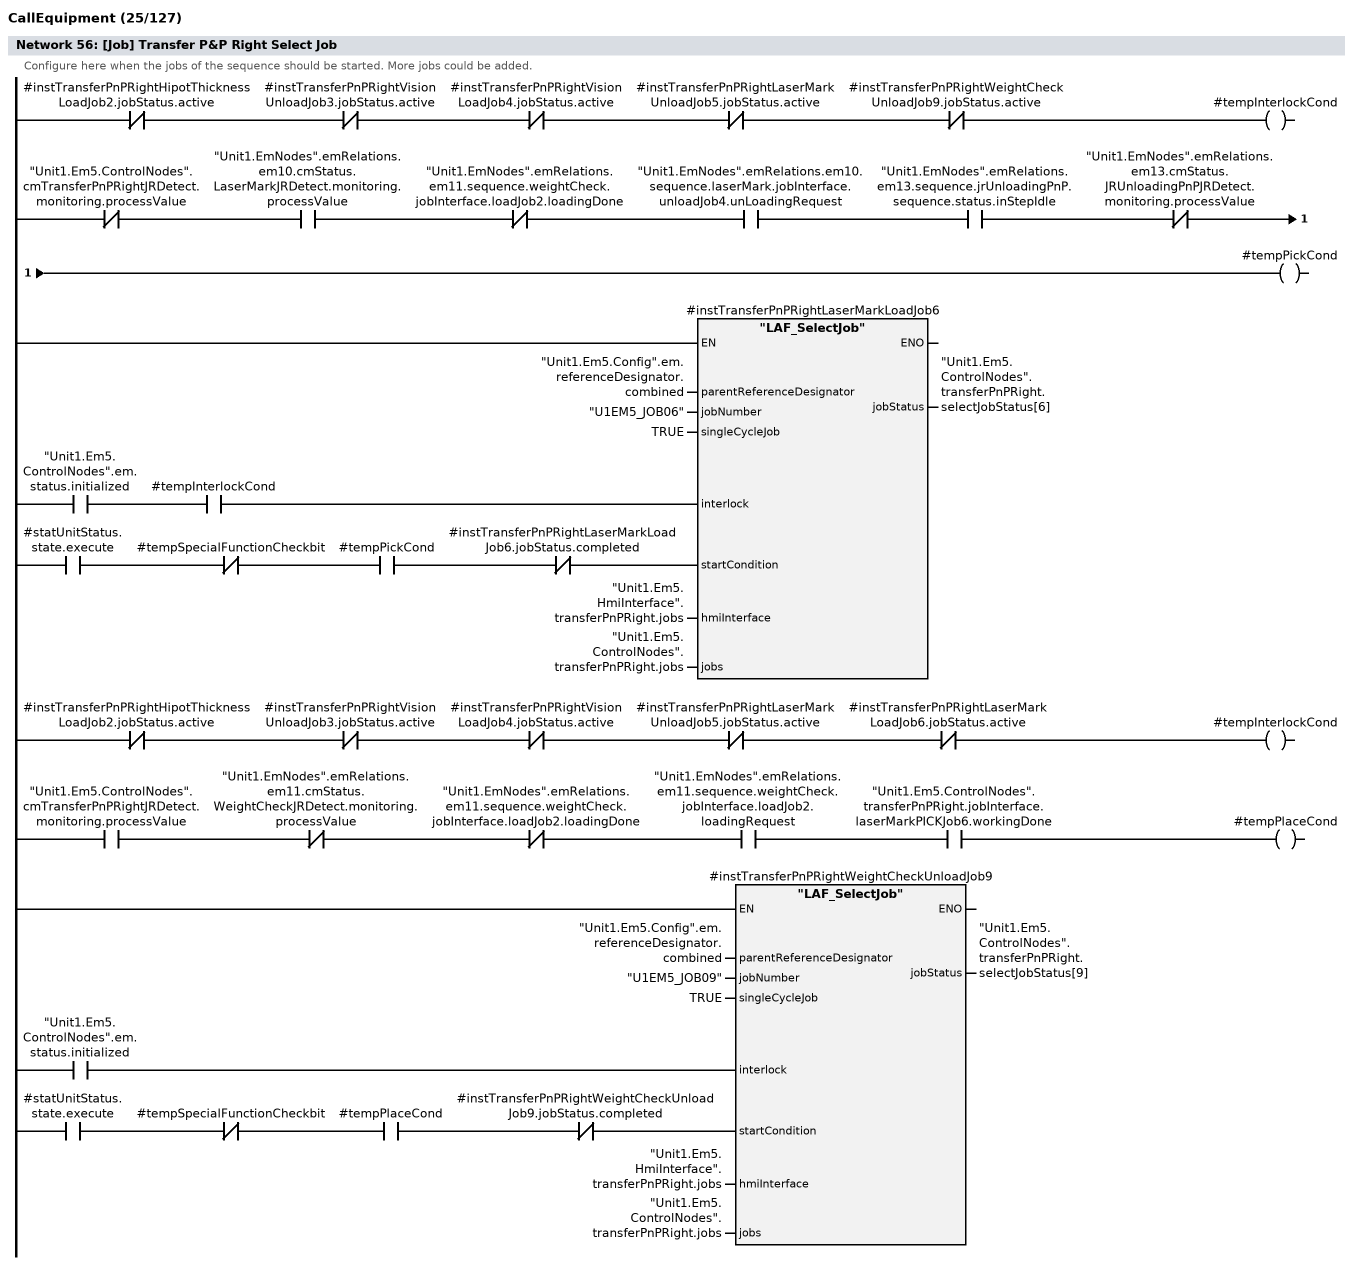
   RUNG wire#powerrail
      I_Contact( #instTransferPnPRightHipotThicknessLoadJob2.jobStatus.active )
      I_Contact( #instTransferPnPRightVisionUnloadJob3.jobStatus.active )
      I_Contact( #instTransferPnPRightVisionLoadJob4.jobStatus.active )
      I_Contact( #instTransferPnPRightLaserMarkUnloadJob5.jobStatus.active )
      I_Contact( #instTransferPnPRightWeightCheckUnloadJob9.jobStatus.active )
      Coil( #tempInterlockCond )
   END_RUNG
   RUNG wire#powerrail
      I_Contact( "Unit1.Em5.ControlNodes".cmTransferPnPRightJRDetect.monitoring.processValue )
      Contact( "Unit1.EmNodes".emRelations.em10.cmStatus.LaserMarkJRDetect.monitoring.processValue )
      I_Contact( "Unit1.EmNodes".emRelations.em11.sequence.weightCheck.jobInterface.loadJob2.loadingDone )
      Contact( "Unit1.EmNodes".emRelations.em10.sequence.laserMark.jobInterface.unloadJob4.unLoadingRequest )
      Contact( "Unit1.EmNodes".emRelations.em13.sequence.jrUnloadingPnP.sequence.status.inStepIdle )
      I_Contact( "Unit1.EmNodes".emRelations.em13.cmStatus.JRUnloadingPnPJRDetect.monitoring.processValue )
      Coil( #tempPickCond )
   END_RUNG
   RUNG wire#powerrail
      #instTransferPnPRightLaserMarkLoadJob6(interlock := wire#w1, startCondition := wire#w2, parentReferenceDesignator := "Unit1.Em5.Config".em.referenceDesignator.combined, jobNumber := "U1EM5_JOB06", singleCycleJob := TRUE, hmiInterface := "Unit1.Em5.HmiInterface".transferPnPRight.jobs, jobs := "Unit1.Em5.ControlNodes".transferPnPRight.jobs, jobStatus => "Unit1.Em5.ControlNodes".transferPnPRight.selectJobStatus[6])
   END_RUNG
   RUNG wire#powerrail
      Contact( "Unit1.Em5.ControlNodes".em.status.initialized )
      Contact( #tempInterlockCond )
   END_RUNG wire#w1
   RUNG wire#powerrail
      Contact( #statUnitStatus.state.execute )
      I_Contact( #tempSpecialFunctionCheckbit )
      Contact( #tempPickCond )
      I_Contact( #instTransferPnPRightLaserMarkLoadJob6.jobStatus.completed )
   END_RUNG wire#w2
   RUNG wire#powerrail
      I_Contact( #instTransferPnPRightHipotThicknessLoadJob2.jobStatus.active )
      I_Contact( #instTransferPnPRightVisionUnloadJob3.jobStatus.active )
      I_Contact( #instTransferPnPRightVisionLoadJob4.jobStatus.active )
      I_Contact( #instTransferPnPRightLaserMarkUnloadJob5.jobStatus.active )
      I_Contact( #instTransferPnPRightLaserMarkLoadJob6.jobStatus.active )
      Coil( #tempInterlockCond )
   END_RUNG
   RUNG wire#powerrail
      Contact( "Unit1.Em5.ControlNodes".cmTransferPnPRightJRDetect.monitoring.processValue )
      I_Contact( "Unit1.EmNodes".emRelations.em11.cmStatus.WeightCheckJRDetect.monitoring.processValue )
      I_Contact( "Unit1.EmNodes".emRelations.em11.sequence.weightCheck.jobInterface.loadJob2.loadingDone )
      Contact( "Unit1.EmNodes".emRelations.em11.sequence.weightCheck.jobInterface.loadJob2.loadingRequest )
      Contact( "Unit1.Em5.ControlNodes".transferPnPRight.jobInterface.laserMarkPICKJob6.workingDone )
      Coil( #tempPlaceCond )
   END_RUNG
   RUNG wire#powerrail
      #instTransferPnPRightWeightCheckUnloadJob9(interlock := wire#w3, startCondition := wire#w4, parentReferenceDesignator := "Unit1.Em5.Config".em.referenceDesignator.combined, jobNumber := "U1EM5_JOB09", singleCycleJob := TRUE, hmiInterface := "Unit1.Em5.HmiInterface".transferPnPRight.jobs, jobs := "Unit1.Em5.ControlNodes".transferPnPRight.jobs, jobStatus => "Unit1.Em5.ControlNodes".transferPnPRight.selectJobStatus[9])
   END_RUNG
   RUNG wire#powerrail
      Contact( "Unit1.Em5.ControlNodes".em.status.initialized )
   END_RUNG wire#w3
   RUNG wire#powerrail
      Contact( #statUnitStatus.state.execute )
      I_Contact( #tempSpecialFunctionCheckbit )
      Contact( #tempPlaceCond )
      I_Contact( #instTransferPnPRightWeightCheckUnloadJob9.jobStatus.completed )
   END_RUNG wire#w4
   // the same network as SCL:
   #tempInterlockCond := NOT #instTransferPnPRightHipotThicknessLoadJob2.jobStatus.active AND NOT #instTransferPnPRightVisionUnloadJob3.jobStatus.active AND NOT #instTransferPnPRightVisionLoadJob4.jobStatus.active AND NOT #instTransferPnPRightLaserMarkUnloadJob5.jobStatus.active AND NOT #instTransferPnPRightWeightCheckUnloadJob9.jobStatus.active;
   #tempPickCond := NOT "Unit1.Em5.ControlNodes".cmTransferPnPRightJRDetect.monitoring.processValue AND "Unit1.EmNodes".emRelations.em10.cmStatus.LaserMarkJRDetect.monitoring.processValue AND NOT "Unit1.EmNodes".emRelations.em11.sequence.weightCheck.jobInterface.loadJob2.loadingDone AND "Unit1.EmNodes".emRelations.em10.sequence.laserMark.jobInterface.unloadJob4.unLoadingRequest AND "Unit1.EmNodes".emRelations.em13.sequence.jrUnloadingPnP.sequence.status.inStepIdle AND NOT "Unit1.EmNodes".emRelations.em13.cmStatus.JRUnloadingPnPJRDetect.monitoring.processValue;
   #instTransferPnPRightLaserMarkLoadJob6(parentReferenceDesignator := "Unit1.Em5.Config".em.referenceDesignator.combined,   // "LAF_SelectJob"
                           jobNumber := "U1EM5_JOB06",
                           singleCycleJob := TRUE,
                           interlock := "Unit1.Em5.ControlNodes".em.status.initialized AND #tempInterlockCond,
                           startCondition := #statUnitStatus.state.execute AND NOT #tempSpecialFunctionCheckbit AND #tempPickCond AND NOT #instTransferPnPRightLaserMarkLoadJob6.jobStatus.completed,
                           hmiInterface := "Unit1.Em5.HmiInterface".transferPnPRight.jobs,
                           jobs := "Unit1.Em5.ControlNodes".transferPnPRight.jobs,
                           jobStatus => "Unit1.Em5.ControlNodes".transferPnPRight.selectJobStatus[6]);
   #tempInterlockCond := NOT #instTransferPnPRightHipotThicknessLoadJob2.jobStatus.active AND NOT #instTransferPnPRightVisionUnloadJob3.jobStatus.active AND NOT #instTransferPnPRightVisionLoadJob4.jobStatus.active AND NOT #instTransferPnPRightLaserMarkUnloadJob5.jobStatus.active AND NOT #instTransferPnPRightLaserMarkLoadJob6.jobStatus.active;
   #tempPlaceCond := "Unit1.Em5.ControlNodes".cmTransferPnPRightJRDetect.monitoring.processValue AND NOT "Unit1.EmNodes".emRelations.em11.cmStatus.WeightCheckJRDetect.monitoring.processValue AND NOT "Unit1.EmNodes".emRelations.em11.sequence.weightCheck.jobInterface.loadJob2.loadingDone AND "Unit1.EmNodes".emRelations.em11.sequence.weightCheck.jobInterface.loadJob2.loadingRequest AND "Unit1.Em5.ControlNodes".transferPnPRight.jobInterface.laserMarkPICKJob6.workingDone;
   #instTransferPnPRightWeightCheckUnloadJob9(parentReferenceDesignator := "Unit1.Em5.Config".em.referenceDesignator.combined,   // "LAF_SelectJob"
                           jobNumber := "U1EM5_JOB09",
                           singleCycleJob := TRUE,
                           interlock := "Unit1.Em5.ControlNodes".em.status.initialized,
                           startCondition := #statUnitStatus.state.execute AND NOT #tempSpecialFunctionCheckbit AND #tempPlaceCond AND NOT #instTransferPnPRightWeightCheckUnloadJob9.jobStatus.completed,
                           hmiInterface := "Unit1.Em5.HmiInterface".transferPnPRight.jobs,
                           jobs := "Unit1.Em5.ControlNodes".transferPnPRight.jobs,
                           jobStatus => "Unit1.Em5.ControlNodes".transferPnPRight.selectJobStatus[9]);
END_REGION

REGION Network 57: Transfer P&P Right Job Interface [Laser Loading]
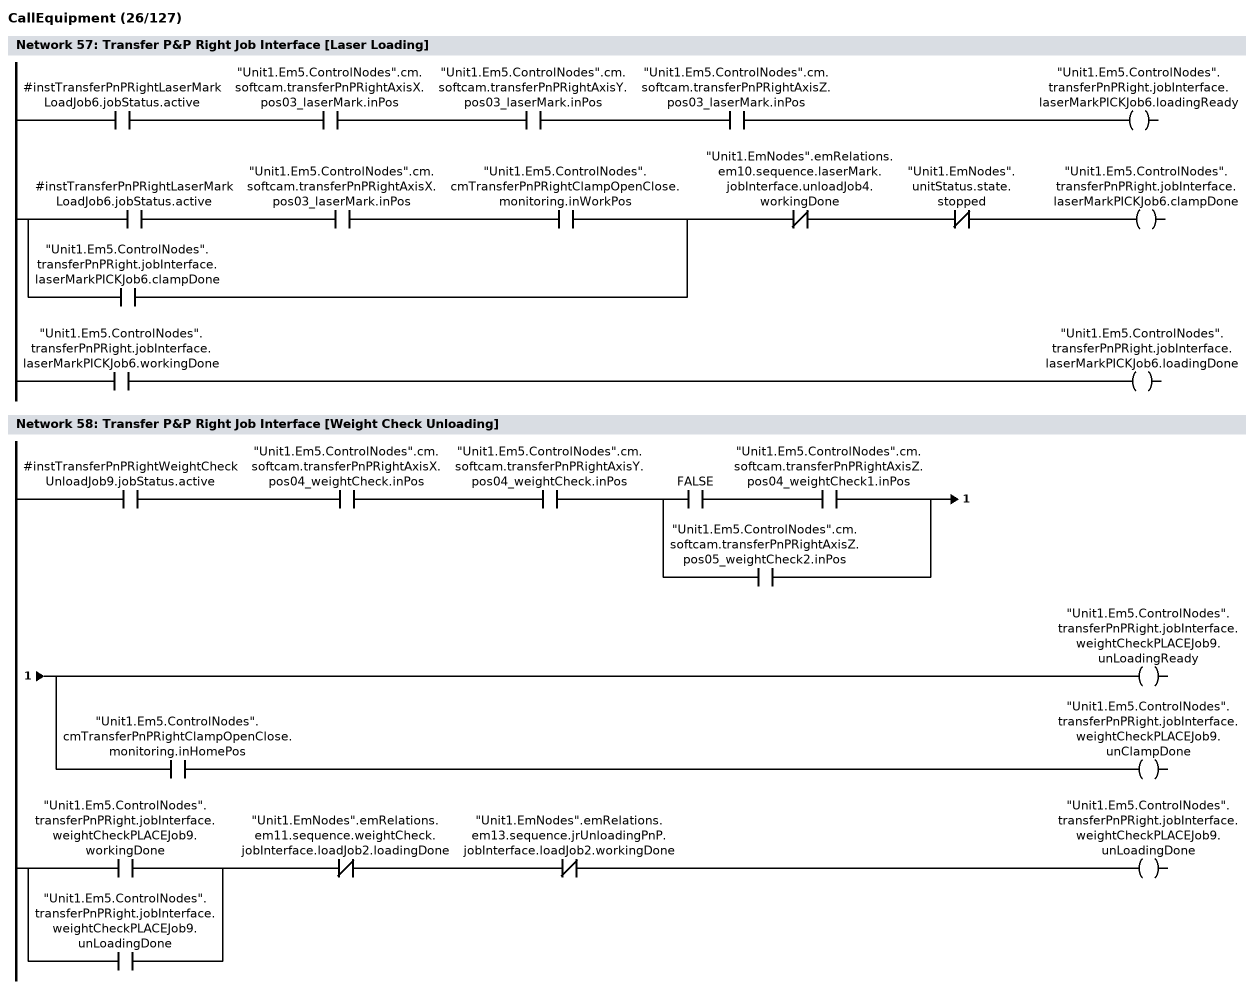
   RUNG wire#powerrail
      Contact( #instTransferPnPRightLaserMarkLoadJob6.jobStatus.active )
      Contact( "Unit1.Em5.ControlNodes".cm.softcam.transferPnPRightAxisX.pos03_laserMark.inPos )
      Contact( "Unit1.Em5.ControlNodes".cm.softcam.transferPnPRightAxisY.pos03_laserMark.inPos )
      Contact( "Unit1.Em5.ControlNodes".cm.softcam.transferPnPRightAxisZ.pos03_laserMark.inPos )
      Coil( "Unit1.Em5.ControlNodes".transferPnPRight.jobInterface.laserMarkPICKJob6.loadingReady )
   END_RUNG
   RUNG wire#powerrail
      Contact( #instTransferPnPRightLaserMarkLoadJob6.jobStatus.active )
      Contact( "Unit1.Em5.ControlNodes".cm.softcam.transferPnPRightAxisX.pos03_laserMark.inPos )
      Contact( "Unit1.Em5.ControlNodes".cmTransferPnPRightClampOpenClose.monitoring.inWorkPos )
      wire#w1
      I_Contact( "Unit1.EmNodes".emRelations.em10.sequence.laserMark.jobInterface.unloadJob4.workingDone )
      I_Contact( "Unit1.EmNodes".unitStatus.state.stopped )
      Coil( "Unit1.Em5.ControlNodes".transferPnPRight.jobInterface.laserMarkPICKJob6.clampDone )
   END_RUNG
   RUNG wire#powerrail
      Contact( "Unit1.Em5.ControlNodes".transferPnPRight.jobInterface.laserMarkPICKJob6.clampDone )
   END_RUNG wire#w1
   RUNG wire#powerrail
      Contact( "Unit1.Em5.ControlNodes".transferPnPRight.jobInterface.laserMarkPICKJob6.workingDone )
      Coil( "Unit1.Em5.ControlNodes".transferPnPRight.jobInterface.laserMarkPICKJob6.loadingDone )
   END_RUNG
   // the same network as SCL:
   "Unit1.Em5.ControlNodes".transferPnPRight.jobInterface.laserMarkPICKJob6.loadingReady := #instTransferPnPRightLaserMarkLoadJob6.jobStatus.active AND "Unit1.Em5.ControlNodes".cm.softcam.transferPnPRightAxisX.pos03_laserMark.inPos AND "Unit1.Em5.ControlNodes".cm.softcam.transferPnPRightAxisY.pos03_laserMark.inPos AND "Unit1.Em5.ControlNodes".cm.softcam.transferPnPRightAxisZ.pos03_laserMark.inPos;
   "Unit1.Em5.ControlNodes".transferPnPRight.jobInterface.laserMarkPICKJob6.clampDone := ((#instTransferPnPRightLaserMarkLoadJob6.jobStatus.active AND "Unit1.Em5.ControlNodes".cm.softcam.transferPnPRightAxisX.pos03_laserMark.inPos AND "Unit1.Em5.ControlNodes".cmTransferPnPRightClampOpenClose.monitoring.inWorkPos) OR "Unit1.Em5.ControlNodes".transferPnPRight.jobInterface.laserMarkPICKJob6.clampDone) AND NOT "Unit1.EmNodes".emRelations.em10.sequence.laserMark.jobInterface.unloadJob4.workingDone AND NOT "Unit1.EmNodes".unitStatus.state.stopped;
   "Unit1.Em5.ControlNodes".transferPnPRight.jobInterface.laserMarkPICKJob6.loadingDone := "Unit1.Em5.ControlNodes".transferPnPRight.jobInterface.laserMarkPICKJob6.workingDone;
END_REGION

REGION Network 58: Transfer P&P Right Job Interface [Weight Check Unloading]
   RUNG wire#powerrail
      Contact( #instTransferPnPRightWeightCheckUnloadJob9.jobStatus.active )
      Contact( "Unit1.Em5.ControlNodes".cm.softcam.transferPnPRightAxisX.pos04_weightCheck.inPos )
      Contact( "Unit1.Em5.ControlNodes".cm.softcam.transferPnPRightAxisY.pos04_weightCheck.inPos )
      wire#w1
      Contact( FALSE )
      Contact( "Unit1.Em5.ControlNodes".cm.softcam.transferPnPRightAxisZ.pos04_weightCheck1.inPos )
      wire#w2
      Coil( "Unit1.Em5.ControlNodes".transferPnPRight.jobInterface.weightCheckPLACEJob9.unLoadingReady )
   END_RUNG
   RUNG wire#w1
      Contact( "Unit1.Em5.ControlNodes".cm.softcam.transferPnPRightAxisZ.pos05_weightCheck2.inPos )
   END_RUNG wire#w2
   RUNG wire#w2
      Contact( "Unit1.Em5.ControlNodes".cmTransferPnPRightClampOpenClose.monitoring.inHomePos )
      Coil( "Unit1.Em5.ControlNodes".transferPnPRight.jobInterface.weightCheckPLACEJob9.unClampDone )
   END_RUNG
   RUNG wire#powerrail
      Contact( "Unit1.Em5.ControlNodes".transferPnPRight.jobInterface.weightCheckPLACEJob9.workingDone )
      wire#w3
      I_Contact( "Unit1.EmNodes".emRelations.em11.sequence.weightCheck.jobInterface.loadJob2.loadingDone )
      I_Contact( "Unit1.EmNodes".emRelations.em13.sequence.jrUnloadingPnP.jobInterface.loadJob2.workingDone )
      Coil( "Unit1.Em5.ControlNodes".transferPnPRight.jobInterface.weightCheckPLACEJob9.unLoadingDone )
   END_RUNG
   RUNG wire#powerrail
      Contact( "Unit1.Em5.ControlNodes".transferPnPRight.jobInterface.weightCheckPLACEJob9.unLoadingDone )
   END_RUNG wire#w3
   // the same network as SCL:
   "Unit1.Em5.ControlNodes".transferPnPRight.jobInterface.weightCheckPLACEJob9.unLoadingReady := #instTransferPnPRightWeightCheckUnloadJob9.jobStatus.active AND "Unit1.Em5.ControlNodes".cm.softcam.transferPnPRightAxisX.pos04_weightCheck.inPos AND "Unit1.Em5.ControlNodes".cm.softcam.transferPnPRightAxisY.pos04_weightCheck.inPos AND ((FALSE AND "Unit1.Em5.ControlNodes".cm.softcam.transferPnPRightAxisZ.pos04_weightCheck1.inPos) OR "Unit1.Em5.ControlNodes".cm.softcam.transferPnPRightAxisZ.pos05_weightCheck2.inPos);
   "Unit1.Em5.ControlNodes".transferPnPRight.jobInterface.weightCheckPLACEJob9.unClampDone := "Unit1.Em5.ControlNodes".transferPnPRight.jobInterface.weightCheckPLACEJob9.unLoadingReady AND "Unit1.Em5.ControlNodes".cmTransferPnPRightClampOpenClose.monitoring.inHomePos;
   "Unit1.Em5.ControlNodes".transferPnPRight.jobInterface.weightCheckPLACEJob9.unLoadingDone := ("Unit1.Em5.ControlNodes".transferPnPRight.jobInterface.weightCheckPLACEJob9.workingDone OR "Unit1.Em5.ControlNodes".transferPnPRight.jobInterface.weightCheckPLACEJob9.unLoadingDone) AND NOT "Unit1.EmNodes".emRelations.em11.sequence.weightCheck.jobInterface.loadJob2.loadingDone AND NOT "Unit1.EmNodes".emRelations.em13.sequence.jrUnloadingPnP.jobInterface.loadJob2.workingDone;
END_REGION

REGION Network 59: Transfer P&P Right Job Interface Working Done [Laser Mark → Weight Check]
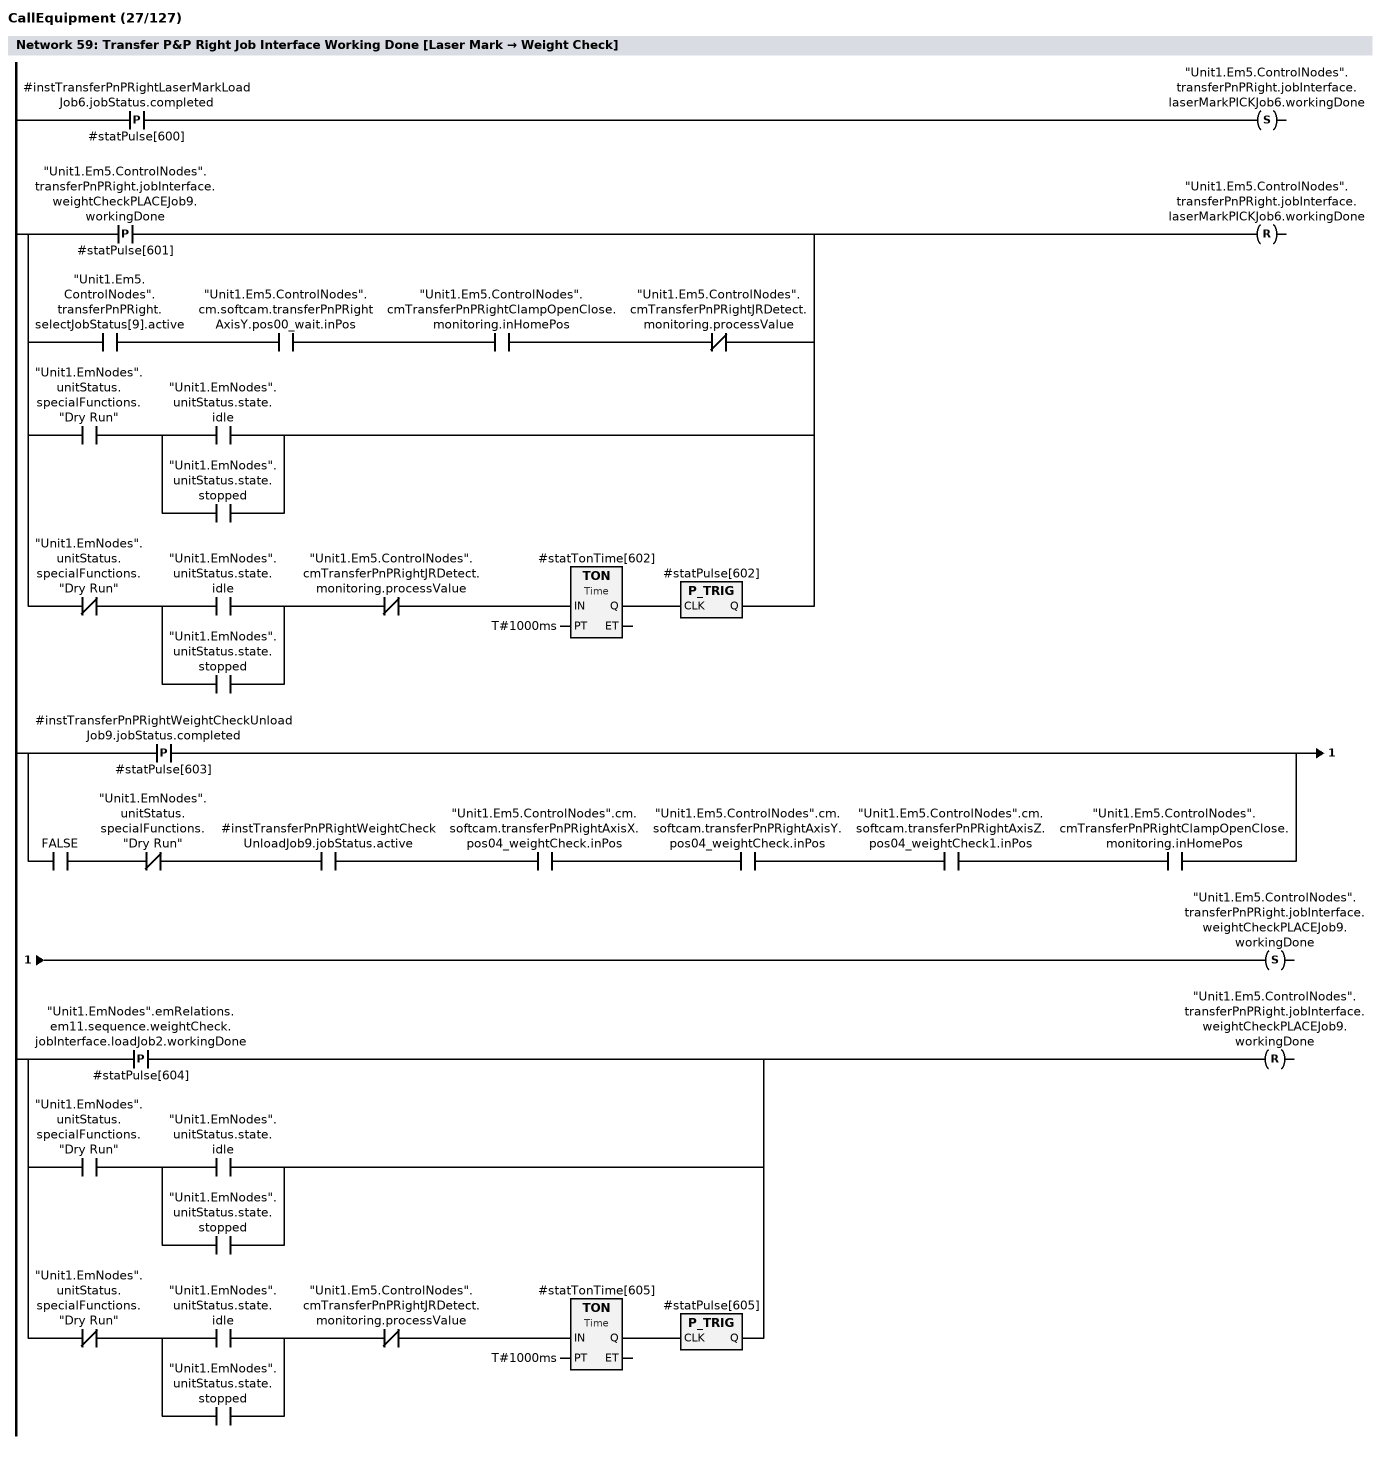
   RUNG wire#powerrail
      P_Contact(operand := #instTransferPnPRightLaserMarkLoadJob6.jobStatus.completed, bit := #statPulse[600])
      S_Coil( "Unit1.Em5.ControlNodes".transferPnPRight.jobInterface.laserMarkPICKJob6.workingDone )
   END_RUNG
   RUNG wire#powerrail
      P_Contact(operand := "Unit1.Em5.ControlNodes".transferPnPRight.jobInterface.weightCheckPLACEJob9.workingDone, bit := #statPulse[601])
      wire#w1
      R_Coil( "Unit1.Em5.ControlNodes".transferPnPRight.jobInterface.laserMarkPICKJob6.workingDone )
   END_RUNG
   RUNG wire#powerrail
      Contact( "Unit1.Em5.ControlNodes".transferPnPRight.selectJobStatus[9].active )
      Contact( "Unit1.Em5.ControlNodes".cm.softcam.transferPnPRightAxisY.pos00_wait.inPos )
      Contact( "Unit1.Em5.ControlNodes".cmTransferPnPRightClampOpenClose.monitoring.inHomePos )
      I_Contact( "Unit1.Em5.ControlNodes".cmTransferPnPRightJRDetect.monitoring.processValue )
   END_RUNG wire#w1
   RUNG wire#powerrail
      Contact( "Unit1.EmNodes".unitStatus.specialFunctions."Dry Run" )
      wire#w2
      Contact( "Unit1.EmNodes".unitStatus.state.idle )
   END_RUNG wire#w1
   RUNG wire#w2
      Contact( "Unit1.EmNodes".unitStatus.state.stopped )
   END_RUNG wire#w1
   RUNG wire#powerrail
      I_Contact( "Unit1.EmNodes".unitStatus.specialFunctions."Dry Run" )
      wire#w3
      Contact( "Unit1.EmNodes".unitStatus.state.idle )
      wire#w4
      I_Contact( "Unit1.Em5.ControlNodes".cmTransferPnPRightJRDetect.monitoring.processValue )
      { S7_Templates := "time_type := Time" } #statTonTime[602].TON(pt := T#1000ms, et =>)
      P_Trig( #statPulse[602] )
   END_RUNG wire#w1
   RUNG wire#w3
      Contact( "Unit1.EmNodes".unitStatus.state.stopped )
   END_RUNG wire#w4
   RUNG wire#powerrail
      P_Contact(operand := #instTransferPnPRightWeightCheckUnloadJob9.jobStatus.completed, bit := #statPulse[603])
      wire#w5
      S_Coil( "Unit1.Em5.ControlNodes".transferPnPRight.jobInterface.weightCheckPLACEJob9.workingDone )
   END_RUNG
   RUNG wire#powerrail
      Contact( FALSE )
      I_Contact( "Unit1.EmNodes".unitStatus.specialFunctions."Dry Run" )
      Contact( #instTransferPnPRightWeightCheckUnloadJob9.jobStatus.active )
      Contact( "Unit1.Em5.ControlNodes".cm.softcam.transferPnPRightAxisX.pos04_weightCheck.inPos )
      Contact( "Unit1.Em5.ControlNodes".cm.softcam.transferPnPRightAxisY.pos04_weightCheck.inPos )
      Contact( "Unit1.Em5.ControlNodes".cm.softcam.transferPnPRightAxisZ.pos04_weightCheck1.inPos )
      Contact( "Unit1.Em5.ControlNodes".cmTransferPnPRightClampOpenClose.monitoring.inHomePos )
   END_RUNG wire#w5
   RUNG wire#powerrail
      P_Contact(operand := "Unit1.EmNodes".emRelations.em11.sequence.weightCheck.jobInterface.loadJob2.workingDone, bit := #statPulse[604])
      wire#w6
      R_Coil( "Unit1.Em5.ControlNodes".transferPnPRight.jobInterface.weightCheckPLACEJob9.workingDone )
   END_RUNG
   RUNG wire#powerrail
      Contact( "Unit1.EmNodes".unitStatus.specialFunctions."Dry Run" )
      wire#w7
      Contact( "Unit1.EmNodes".unitStatus.state.idle )
   END_RUNG wire#w6
   RUNG wire#w7
      Contact( "Unit1.EmNodes".unitStatus.state.stopped )
   END_RUNG wire#w6
   RUNG wire#powerrail
      I_Contact( "Unit1.EmNodes".unitStatus.specialFunctions."Dry Run" )
      wire#w8
      Contact( "Unit1.EmNodes".unitStatus.state.idle )
      wire#w9
      I_Contact( "Unit1.Em5.ControlNodes".cmTransferPnPRightJRDetect.monitoring.processValue )
      { S7_Templates := "time_type := Time" } #statTonTime[605].TON(pt := T#1000ms, et =>)
      P_Trig( #statPulse[605] )
   END_RUNG wire#w6
   RUNG wire#w8
      Contact( "Unit1.EmNodes".unitStatus.state.stopped )
   END_RUNG wire#w9
   // the same network as SCL:
   #_w1 := #instTransferPnPRightLaserMarkLoadJob6.jobStatus.completed AND NOT #statPulse[600];   // rising edge of #instTransferPnPRightLaserMarkLoadJob6.jobStatus.completed
   #statPulse[600] := #instTransferPnPRightLaserMarkLoadJob6.jobStatus.completed;
   IF #_w1 THEN
       "Unit1.Em5.ControlNodes".transferPnPRight.jobInterface.laserMarkPICKJob6.workingDone := TRUE;
   END_IF;
   #_w2 := "Unit1.Em5.ControlNodes".transferPnPRight.jobInterface.weightCheckPLACEJob9.workingDone AND NOT #statPulse[601];   // rising edge of "Unit1.Em5.ControlNodes".transferPnPRight.jobInterface.weightCheckPLACEJob9.workingDone
   #statPulse[601] := "Unit1.Em5.ControlNodes".transferPnPRight.jobInterface.weightCheckPLACEJob9.workingDone;
   #statTonTime[602].TON(IN := NOT "Unit1.EmNodes".unitStatus.specialFunctions."Dry Run" AND ("Unit1.EmNodes".unitStatus.state.idle OR "Unit1.EmNodes".unitStatus.state.stopped) AND NOT "Unit1.Em5.ControlNodes".cmTransferPnPRightJRDetect.monitoring.processValue,
                         PT := T#1000ms);
   #_w3 := #statTonTime[602].Q AND NOT #statPulse[602];   // rising edge
   #statPulse[602] := #statTonTime[602].Q;
   IF #_w2 OR ("Unit1.Em5.ControlNodes".transferPnPRight.selectJobStatus[9].active AND "Unit1.Em5.ControlNodes".cm.softcam.transferPnPRightAxisY.pos00_wait.inPos AND "Unit1.Em5.ControlNodes".cmTransferPnPRightClampOpenClose.monitoring.inHomePos AND NOT "Unit1.Em5.ControlNodes".cmTransferPnPRightJRDetect.monitoring.processValue) OR ("Unit1.EmNodes".unitStatus.specialFunctions."Dry Run" AND ("Unit1.EmNodes".unitStatus.state.idle OR "Unit1.EmNodes".unitStatus.state.stopped)) OR #_w3 THEN
       "Unit1.Em5.ControlNodes".transferPnPRight.jobInterface.laserMarkPICKJob6.workingDone := FALSE;
   END_IF;
   #_w4 := #instTransferPnPRightWeightCheckUnloadJob9.jobStatus.completed AND NOT #statPulse[603];   // rising edge of #instTransferPnPRightWeightCheckUnloadJob9.jobStatus.completed
   #statPulse[603] := #instTransferPnPRightWeightCheckUnloadJob9.jobStatus.completed;
   IF #_w4 OR (FALSE AND NOT "Unit1.EmNodes".unitStatus.specialFunctions."Dry Run" AND #instTransferPnPRightWeightCheckUnloadJob9.jobStatus.active AND "Unit1.Em5.ControlNodes".cm.softcam.transferPnPRightAxisX.pos04_weightCheck.inPos AND "Unit1.Em5.ControlNodes".cm.softcam.transferPnPRightAxisY.pos04_weightCheck.inPos AND "Unit1.Em5.ControlNodes".cm.softcam.transferPnPRightAxisZ.pos04_weightCheck1.inPos AND "Unit1.Em5.ControlNodes".cmTransferPnPRightClampOpenClose.monitoring.inHomePos) THEN
       "Unit1.Em5.ControlNodes".transferPnPRight.jobInterface.weightCheckPLACEJob9.workingDone := TRUE;
   END_IF;
   #_w5 := "Unit1.EmNodes".emRelations.em11.sequence.weightCheck.jobInterface.loadJob2.workingDone AND NOT #statPulse[604];   // rising edge of "Unit1.EmNodes".emRelations.em11.sequence.weightCheck.jobInterface.loadJob2.workingDone
   #statPulse[604] := "Unit1.EmNodes".emRelations.em11.sequence.weightCheck.jobInterface.loadJob2.workingDone;
   #statTonTime[605].TON(IN := NOT "Unit1.EmNodes".unitStatus.specialFunctions."Dry Run" AND ("Unit1.EmNodes".unitStatus.state.idle OR "Unit1.EmNodes".unitStatus.state.stopped) AND NOT "Unit1.Em5.ControlNodes".cmTransferPnPRightJRDetect.monitoring.processValue,
                         PT := T#1000ms);
   #_w6 := #statTonTime[605].Q AND NOT #statPulse[605];   // rising edge
   #statPulse[605] := #statTonTime[605].Q;
   IF #_w5 OR ("Unit1.EmNodes".unitStatus.specialFunctions."Dry Run" AND ("Unit1.EmNodes".unitStatus.state.idle OR "Unit1.EmNodes".unitStatus.state.stopped)) OR #_w6 THEN
       "Unit1.Em5.ControlNodes".transferPnPRight.jobInterface.weightCheckPLACEJob9.workingDone := FALSE;
   END_IF;
END_REGION

REGION Network 61: [Job]Transfer P&P Gauge R&R Select Job
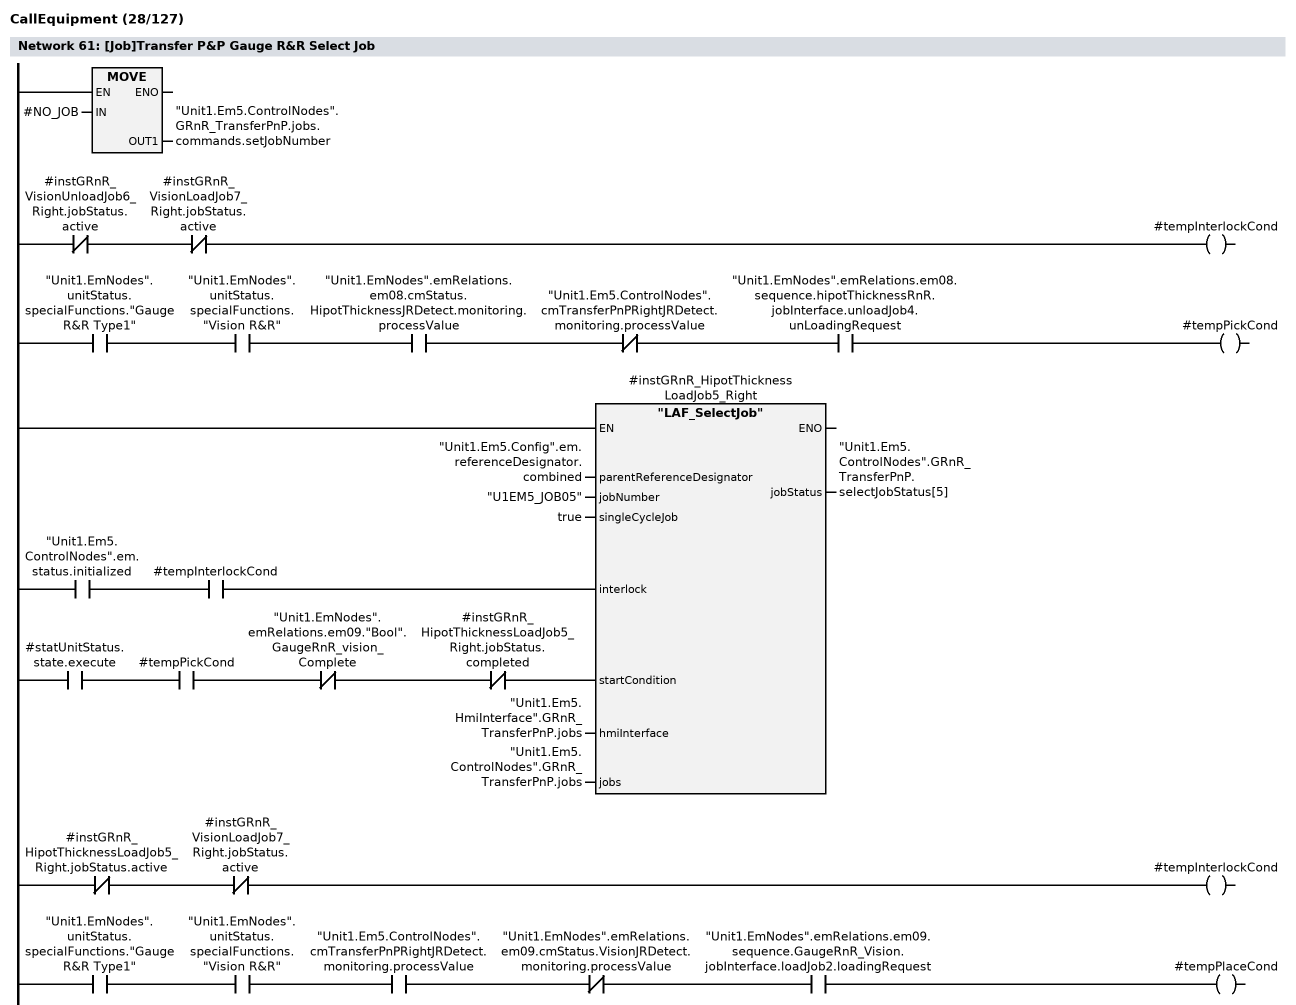
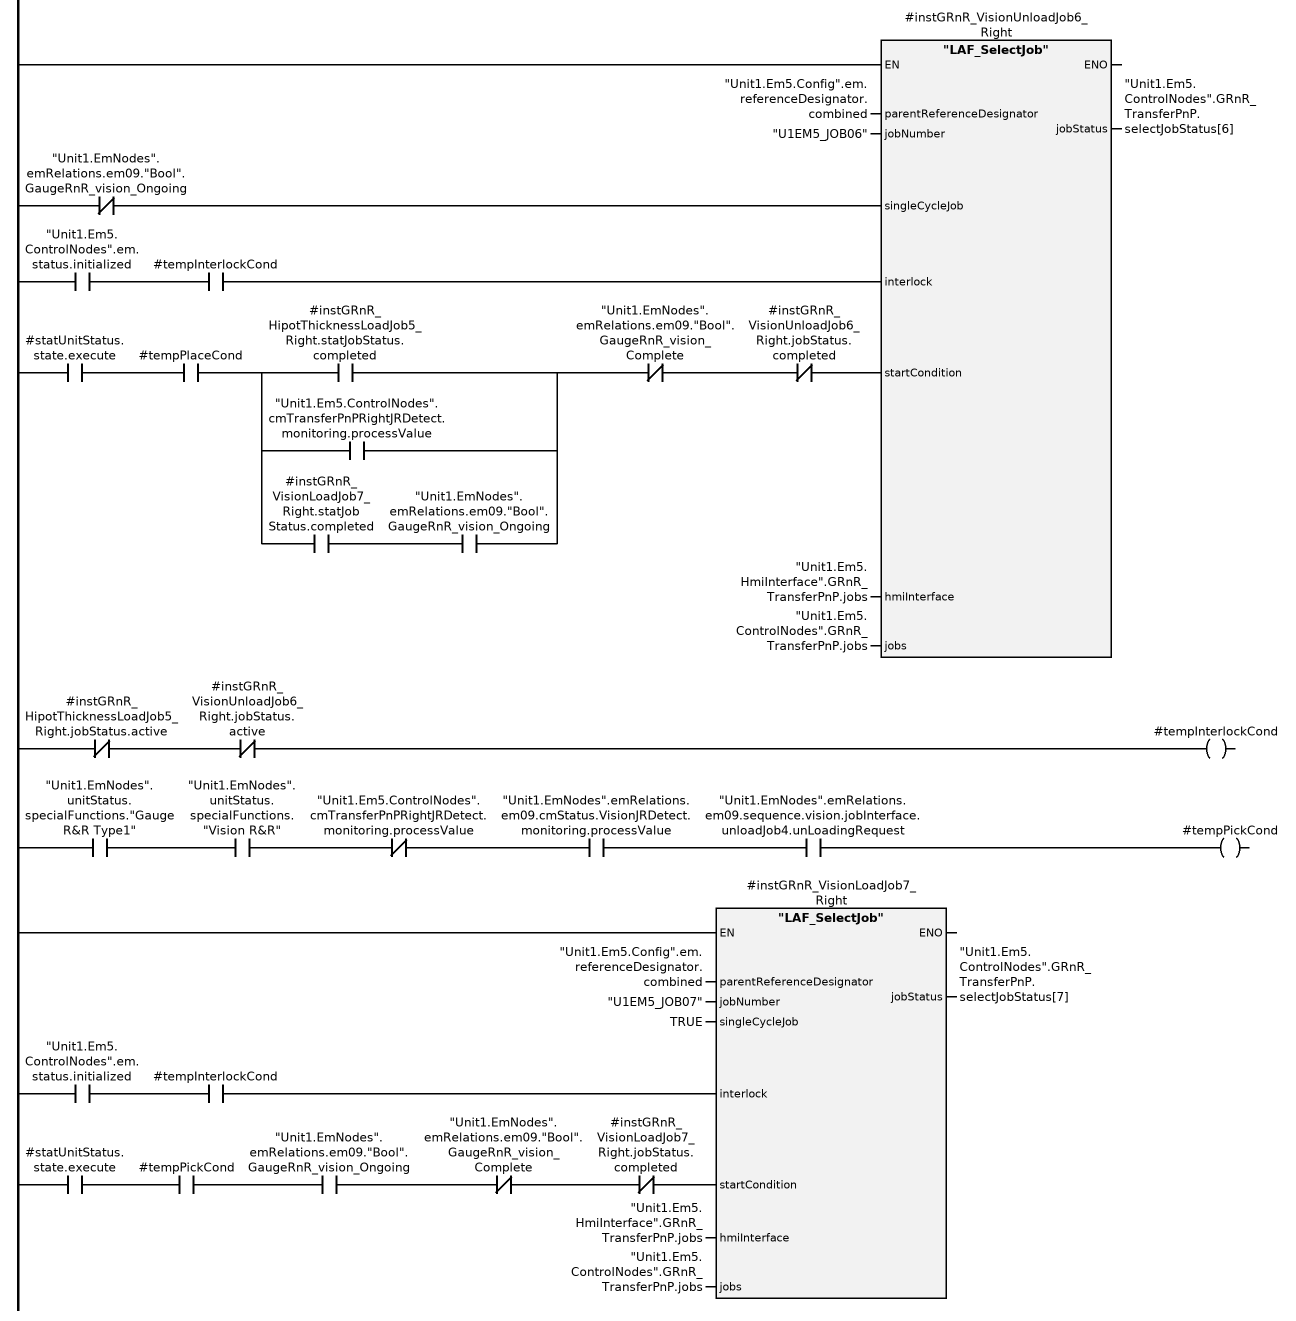
   RUNG wire#powerrail
      Move(in := #NO_JOB, out1 => "Unit1.Em5.ControlNodes".GRnR_TransferPnP.jobs.commands.setJobNumber)
   END_RUNG
   RUNG wire#powerrail
      I_Contact( #instGRnR_VisionUnloadJob6_Right.jobStatus.active )
      I_Contact( #instGRnR_VisionLoadJob7_Right.jobStatus.active )
      Coil( #tempInterlockCond )
   END_RUNG
   RUNG wire#powerrail
      Contact( "Unit1.EmNodes".unitStatus.specialFunctions."Gauge R&R Type1" )
      Contact( "Unit1.EmNodes".unitStatus.specialFunctions."Vision R&R" )
      Contact( "Unit1.EmNodes".emRelations.em08.cmStatus.HipotThicknessJRDetect.monitoring.processValue )
      I_Contact( "Unit1.Em5.ControlNodes".cmTransferPnPRightJRDetect.monitoring.processValue )
      Contact( "Unit1.EmNodes".emRelations.em08.sequence.hipotThicknessRnR.jobInterface.unloadJob4.unLoadingRequest )
      Coil( #tempPickCond )
   END_RUNG
   RUNG wire#powerrail
      #instGRnR_HipotThicknessLoadJob5_Right(interlock := wire#w1, startCondition := wire#w2, parentReferenceDesignator := "Unit1.Em5.Config".em.referenceDesignator.combined, jobNumber := "U1EM5_JOB05", singleCycleJob := true, hmiInterface := "Unit1.Em5.HmiInterface".GRnR_TransferPnP.jobs, jobs := "Unit1.Em5.ControlNodes".GRnR_TransferPnP.jobs, jobStatus => "Unit1.Em5.ControlNodes".GRnR_TransferPnP.selectJobStatus[5])
   END_RUNG
   RUNG wire#powerrail
      Contact( "Unit1.Em5.ControlNodes".em.status.initialized )
      Contact( #tempInterlockCond )
   END_RUNG wire#w1
   RUNG wire#powerrail
      Contact( #statUnitStatus.state.execute )
      Contact( #tempPickCond )
      I_Contact( "Unit1.EmNodes".emRelations.em09."Bool".GaugeRnR_vision_Complete )
      I_Contact( #instGRnR_HipotThicknessLoadJob5_Right.jobStatus.completed )
   END_RUNG wire#w2
   RUNG wire#powerrail
      I_Contact( #instGRnR_HipotThicknessLoadJob5_Right.jobStatus.active )
      I_Contact( #instGRnR_VisionLoadJob7_Right.jobStatus.active )
      Coil( #tempInterlockCond )
   END_RUNG
   RUNG wire#powerrail
      Contact( "Unit1.EmNodes".unitStatus.specialFunctions."Gauge R&R Type1" )
      Contact( "Unit1.EmNodes".unitStatus.specialFunctions."Vision R&R" )
      Contact( "Unit1.Em5.ControlNodes".cmTransferPnPRightJRDetect.monitoring.processValue )
      I_Contact( "Unit1.EmNodes".emRelations.em09.cmStatus.VisionJRDetect.monitoring.processValue )
      Contact( "Unit1.EmNodes".emRelations.em09.sequence.GaugeRnR_Vision.jobInterface.loadJob2.loadingRequest )
      Coil( #tempPlaceCond )
   END_RUNG
   RUNG wire#powerrail
      #instGRnR_VisionUnloadJob6_Right(singleCycleJob := wire#w3, interlock := wire#w4, startCondition := wire#w7, parentReferenceDesignator := "Unit1.Em5.Config".em.referenceDesignator.combined, jobNumber := "U1EM5_JOB06", hmiInterface := "Unit1.Em5.HmiInterface".GRnR_TransferPnP.jobs, jobs := "Unit1.Em5.ControlNodes".GRnR_TransferPnP.jobs, jobStatus => "Unit1.Em5.ControlNodes".GRnR_TransferPnP.selectJobStatus[6])
   END_RUNG
   RUNG wire#powerrail
      I_Contact( "Unit1.EmNodes".emRelations.em09."Bool".GaugeRnR_vision_Ongoing )
   END_RUNG wire#w3
   RUNG wire#powerrail
      Contact( "Unit1.Em5.ControlNodes".em.status.initialized )
      Contact( #tempInterlockCond )
   END_RUNG wire#w4
   RUNG wire#powerrail
      Contact( #statUnitStatus.state.execute )
      Contact( #tempPlaceCond )
      wire#w5
      Contact( #instGRnR_HipotThicknessLoadJob5_Right.statJobStatus.completed )
      wire#w6
      I_Contact( "Unit1.EmNodes".emRelations.em09."Bool".GaugeRnR_vision_Complete )
      I_Contact( #instGRnR_VisionUnloadJob6_Right.jobStatus.completed )
   END_RUNG wire#w7
   RUNG wire#w5
      Contact( "Unit1.Em5.ControlNodes".cmTransferPnPRightJRDetect.monitoring.processValue )
   END_RUNG wire#w6
   RUNG wire#w5
      Contact( #instGRnR_VisionLoadJob7_Right.statJobStatus.completed )
      Contact( "Unit1.EmNodes".emRelations.em09."Bool".GaugeRnR_vision_Ongoing )
   END_RUNG wire#w6
   RUNG wire#powerrail
      I_Contact( #instGRnR_HipotThicknessLoadJob5_Right.jobStatus.active )
      I_Contact( #instGRnR_VisionUnloadJob6_Right.jobStatus.active )
      Coil( #tempInterlockCond )
   END_RUNG
   RUNG wire#powerrail
      Contact( "Unit1.EmNodes".unitStatus.specialFunctions."Gauge R&R Type1" )
      Contact( "Unit1.EmNodes".unitStatus.specialFunctions."Vision R&R" )
      I_Contact( "Unit1.Em5.ControlNodes".cmTransferPnPRightJRDetect.monitoring.processValue )
      Contact( "Unit1.EmNodes".emRelations.em09.cmStatus.VisionJRDetect.monitoring.processValue )
      Contact( "Unit1.EmNodes".emRelations.em09.sequence.vision.jobInterface.unloadJob4.unLoadingRequest )
      Coil( #tempPickCond )
   END_RUNG
   RUNG wire#powerrail
      #instGRnR_VisionLoadJob7_Right(interlock := wire#w8, startCondition := wire#w9, parentReferenceDesignator := "Unit1.Em5.Config".em.referenceDesignator.combined, jobNumber := "U1EM5_JOB07", singleCycleJob := TRUE, hmiInterface := "Unit1.Em5.HmiInterface".GRnR_TransferPnP.jobs, jobs := "Unit1.Em5.ControlNodes".GRnR_TransferPnP.jobs, jobStatus => "Unit1.Em5.ControlNodes".GRnR_TransferPnP.selectJobStatus[7])
   END_RUNG
   RUNG wire#powerrail
      Contact( "Unit1.Em5.ControlNodes".em.status.initialized )
      Contact( #tempInterlockCond )
   END_RUNG wire#w8
   RUNG wire#powerrail
      Contact( #statUnitStatus.state.execute )
      Contact( #tempPickCond )
      Contact( "Unit1.EmNodes".emRelations.em09."Bool".GaugeRnR_vision_Ongoing )
      I_Contact( "Unit1.EmNodes".emRelations.em09."Bool".GaugeRnR_vision_Complete )
      I_Contact( #instGRnR_VisionLoadJob7_Right.jobStatus.completed )
   END_RUNG wire#w9
   // the same network as SCL:
   "Unit1.Em5.ControlNodes".GRnR_TransferPnP.jobs.commands.setJobNumber := #NO_JOB;
   #tempInterlockCond := NOT #instGRnR_VisionUnloadJob6_Right.jobStatus.active AND NOT #instGRnR_VisionLoadJob7_Right.jobStatus.active;
   #tempPickCond := "Unit1.EmNodes".unitStatus.specialFunctions."Gauge R&R Type1" AND "Unit1.EmNodes".unitStatus.specialFunctions."Vision R&R" AND "Unit1.EmNodes".emRelations.em08.cmStatus.HipotThicknessJRDetect.monitoring.processValue AND NOT "Unit1.Em5.ControlNodes".cmTransferPnPRightJRDetect.monitoring.processValue AND "Unit1.EmNodes".emRelations.em08.sequence.hipotThicknessRnR.jobInterface.unloadJob4.unLoadingRequest;
   #instGRnR_HipotThicknessLoadJob5_Right(parentReferenceDesignator := "Unit1.Em5.Config".em.referenceDesignator.combined,   // "LAF_SelectJob"
                           jobNumber := "U1EM5_JOB05",
                           singleCycleJob := true,
                           interlock := "Unit1.Em5.ControlNodes".em.status.initialized AND #tempInterlockCond,
                           startCondition := #statUnitStatus.state.execute AND #tempPickCond AND NOT "Unit1.EmNodes".emRelations.em09."Bool".GaugeRnR_vision_Complete AND NOT #instGRnR_HipotThicknessLoadJob5_Right.jobStatus.completed,
                           hmiInterface := "Unit1.Em5.HmiInterface".GRnR_TransferPnP.jobs,
                           jobs := "Unit1.Em5.ControlNodes".GRnR_TransferPnP.jobs,
                           jobStatus => "Unit1.Em5.ControlNodes".GRnR_TransferPnP.selectJobStatus[5]);
   #tempInterlockCond := NOT #instGRnR_HipotThicknessLoadJob5_Right.jobStatus.active AND NOT #instGRnR_VisionLoadJob7_Right.jobStatus.active;
   #tempPlaceCond := "Unit1.EmNodes".unitStatus.specialFunctions."Gauge R&R Type1" AND "Unit1.EmNodes".unitStatus.specialFunctions."Vision R&R" AND "Unit1.Em5.ControlNodes".cmTransferPnPRightJRDetect.monitoring.processValue AND NOT "Unit1.EmNodes".emRelations.em09.cmStatus.VisionJRDetect.monitoring.processValue AND "Unit1.EmNodes".emRelations.em09.sequence.GaugeRnR_Vision.jobInterface.loadJob2.loadingRequest;
   #instGRnR_VisionUnloadJob6_Right(parentReferenceDesignator := "Unit1.Em5.Config".em.referenceDesignator.combined,   // "LAF_SelectJob"
                           jobNumber := "U1EM5_JOB06",
                           singleCycleJob := NOT "Unit1.EmNodes".emRelations.em09."Bool".GaugeRnR_vision_Ongoing,
                           interlock := "Unit1.Em5.ControlNodes".em.status.initialized AND #tempInterlockCond,
                           startCondition := #statUnitStatus.state.execute AND #tempPlaceCond AND (#instGRnR_HipotThicknessLoadJob5_Right.statJobStatus.completed OR "Unit1.Em5.ControlNodes".cmTransferPnPRightJRDetect.monitoring.processValue OR (#instGRnR_VisionLoadJob7_Right.statJobStatus.completed AND "Unit1.EmNodes".emRelations.em09."Bool".GaugeRnR_vision_Ongoing)) AND NOT "Unit1.EmNodes".emRelations.em09."Bool".GaugeRnR_vision_Complete AND NOT #instGRnR_VisionUnloadJob6_Right.jobStatus.completed,
                           hmiInterface := "Unit1.Em5.HmiInterface".GRnR_TransferPnP.jobs,
                           jobs := "Unit1.Em5.ControlNodes".GRnR_TransferPnP.jobs,
                           jobStatus => "Unit1.Em5.ControlNodes".GRnR_TransferPnP.selectJobStatus[6]);
   #tempInterlockCond := NOT #instGRnR_HipotThicknessLoadJob5_Right.jobStatus.active AND NOT #instGRnR_VisionUnloadJob6_Right.jobStatus.active;
   #tempPickCond := "Unit1.EmNodes".unitStatus.specialFunctions."Gauge R&R Type1" AND "Unit1.EmNodes".unitStatus.specialFunctions."Vision R&R" AND NOT "Unit1.Em5.ControlNodes".cmTransferPnPRightJRDetect.monitoring.processValue AND "Unit1.EmNodes".emRelations.em09.cmStatus.VisionJRDetect.monitoring.processValue AND "Unit1.EmNodes".emRelations.em09.sequence.vision.jobInterface.unloadJob4.unLoadingRequest;
   #instGRnR_VisionLoadJob7_Right(parentReferenceDesignator := "Unit1.Em5.Config".em.referenceDesignator.combined,   // "LAF_SelectJob"
                           jobNumber := "U1EM5_JOB07",
                           singleCycleJob := TRUE,
                           interlock := "Unit1.Em5.ControlNodes".em.status.initialized AND #tempInterlockCond,
                           startCondition := #statUnitStatus.state.execute AND #tempPickCond AND "Unit1.EmNodes".emRelations.em09."Bool".GaugeRnR_vision_Ongoing AND NOT "Unit1.EmNodes".emRelations.em09."Bool".GaugeRnR_vision_Complete AND NOT #instGRnR_VisionLoadJob7_Right.jobStatus.completed,
                           hmiInterface := "Unit1.Em5.HmiInterface".GRnR_TransferPnP.jobs,
                           jobs := "Unit1.Em5.ControlNodes".GRnR_TransferPnP.jobs,
                           jobStatus => "Unit1.Em5.ControlNodes".GRnR_TransferPnP.selectJobStatus[7]);
END_REGION

REGION Network 62: Transfer P&P Gague R&R Job Interface [Side Tape Loading][Left]
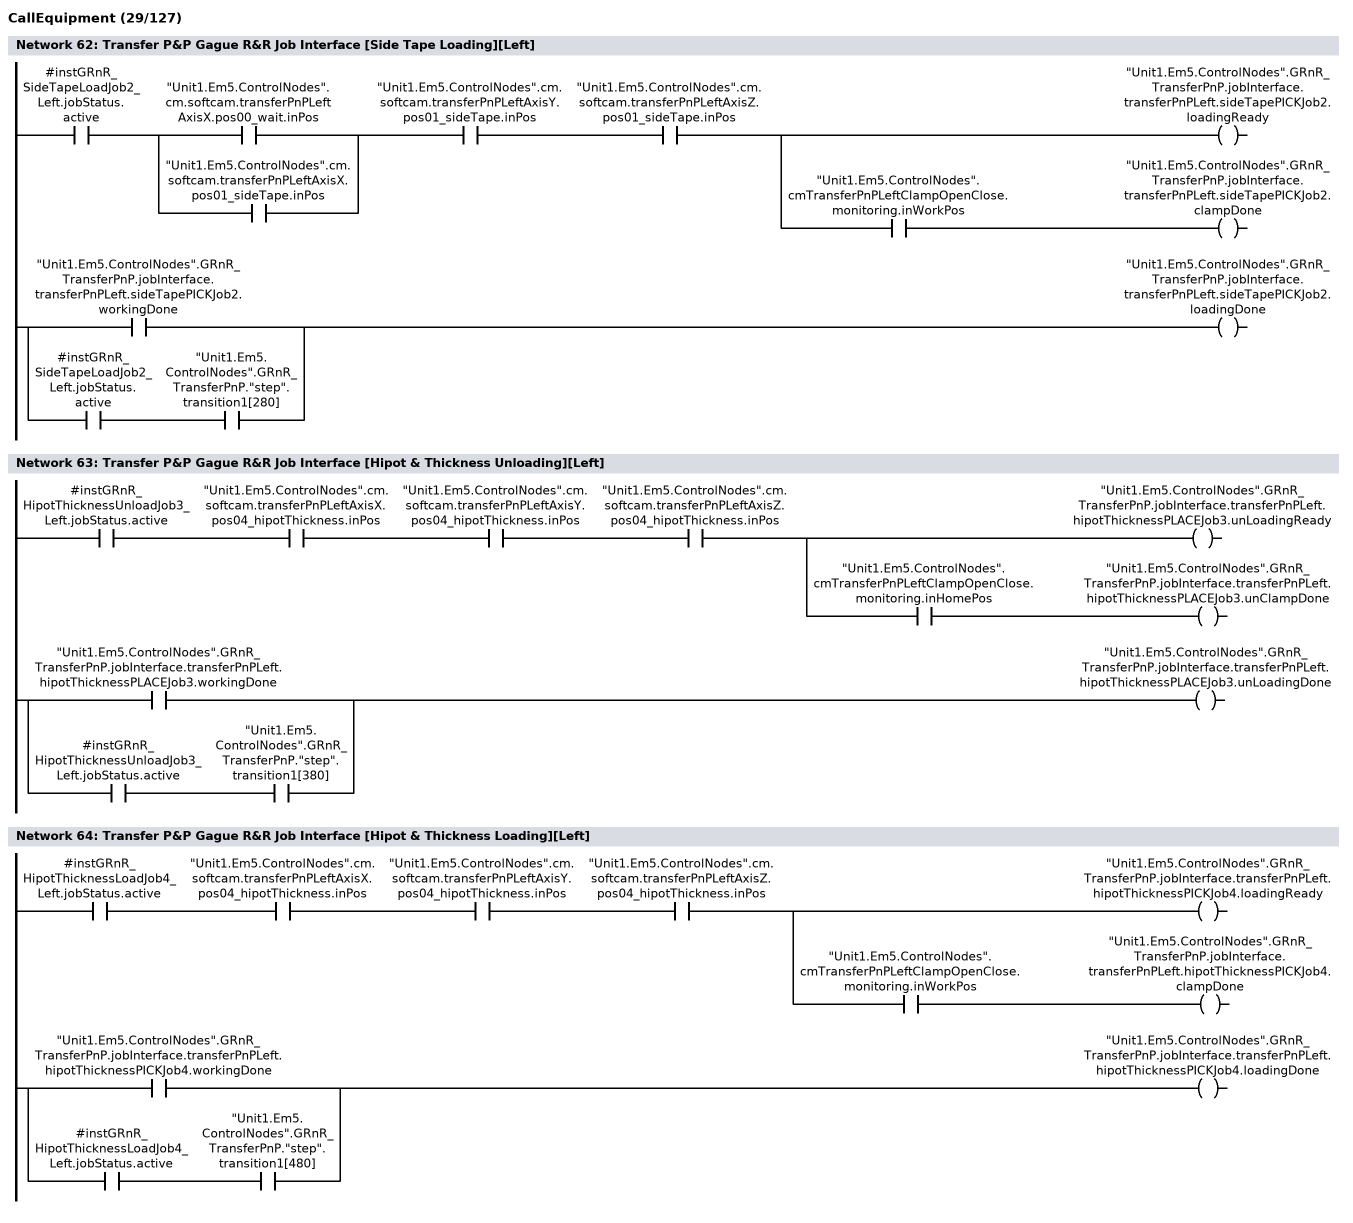
   RUNG wire#powerrail
      Contact( #instGRnR_SideTapeLoadJob2_Left.jobStatus.active )
      wire#w1
      Contact( "Unit1.Em5.ControlNodes".cm.softcam.transferPnPLeftAxisX.pos00_wait.inPos )
      wire#w2
      Contact( "Unit1.Em5.ControlNodes".cm.softcam.transferPnPLeftAxisY.pos01_sideTape.inPos )
      Contact( "Unit1.Em5.ControlNodes".cm.softcam.transferPnPLeftAxisZ.pos01_sideTape.inPos )
      wire#w3
      Coil( "Unit1.Em5.ControlNodes".GRnR_TransferPnP.jobInterface.transferPnPLeft.sideTapePICKJob2.loadingReady )
   END_RUNG
   RUNG wire#w1
      Contact( "Unit1.Em5.ControlNodes".cm.softcam.transferPnPLeftAxisX.pos01_sideTape.inPos )
   END_RUNG wire#w2
   RUNG wire#w3
      Contact( "Unit1.Em5.ControlNodes".cmTransferPnPLeftClampOpenClose.monitoring.inWorkPos )
      Coil( "Unit1.Em5.ControlNodes".GRnR_TransferPnP.jobInterface.transferPnPLeft.sideTapePICKJob2.clampDone )
   END_RUNG
   RUNG wire#powerrail
      Contact( "Unit1.Em5.ControlNodes".GRnR_TransferPnP.jobInterface.transferPnPLeft.sideTapePICKJob2.workingDone )
      wire#w4
      Coil( "Unit1.Em5.ControlNodes".GRnR_TransferPnP.jobInterface.transferPnPLeft.sideTapePICKJob2.loadingDone )
   END_RUNG
   RUNG wire#powerrail
      Contact( #instGRnR_SideTapeLoadJob2_Left.jobStatus.active )
      Contact( "Unit1.Em5.ControlNodes".GRnR_TransferPnP."step".transition1[280] )
   END_RUNG wire#w4
   // the same network as SCL:
   "Unit1.Em5.ControlNodes".GRnR_TransferPnP.jobInterface.transferPnPLeft.sideTapePICKJob2.loadingReady := #instGRnR_SideTapeLoadJob2_Left.jobStatus.active AND ("Unit1.Em5.ControlNodes".cm.softcam.transferPnPLeftAxisX.pos00_wait.inPos OR "Unit1.Em5.ControlNodes".cm.softcam.transferPnPLeftAxisX.pos01_sideTape.inPos) AND "Unit1.Em5.ControlNodes".cm.softcam.transferPnPLeftAxisY.pos01_sideTape.inPos AND "Unit1.Em5.ControlNodes".cm.softcam.transferPnPLeftAxisZ.pos01_sideTape.inPos;
   "Unit1.Em5.ControlNodes".GRnR_TransferPnP.jobInterface.transferPnPLeft.sideTapePICKJob2.clampDone := "Unit1.Em5.ControlNodes".GRnR_TransferPnP.jobInterface.transferPnPLeft.sideTapePICKJob2.loadingReady AND "Unit1.Em5.ControlNodes".cmTransferPnPLeftClampOpenClose.monitoring.inWorkPos;
   "Unit1.Em5.ControlNodes".GRnR_TransferPnP.jobInterface.transferPnPLeft.sideTapePICKJob2.loadingDone := "Unit1.Em5.ControlNodes".GRnR_TransferPnP.jobInterface.transferPnPLeft.sideTapePICKJob2.workingDone OR (#instGRnR_SideTapeLoadJob2_Left.jobStatus.active AND "Unit1.Em5.ControlNodes".GRnR_TransferPnP."step".transition1[280]);
END_REGION

REGION Network 63: Transfer P&P Gague R&R Job Interface [Hipot & Thickness Unloading][Left]
   RUNG wire#powerrail
      Contact( #instGRnR_HipotThicknessUnloadJob3_Left.jobStatus.active )
      Contact( "Unit1.Em5.ControlNodes".cm.softcam.transferPnPLeftAxisX.pos04_hipotThickness.inPos )
      Contact( "Unit1.Em5.ControlNodes".cm.softcam.transferPnPLeftAxisY.pos04_hipotThickness.inPos )
      Contact( "Unit1.Em5.ControlNodes".cm.softcam.transferPnPLeftAxisZ.pos04_hipotThickness.inPos )
      wire#w1
      Coil( "Unit1.Em5.ControlNodes".GRnR_TransferPnP.jobInterface.transferPnPLeft.hipotThicknessPLACEJob3.unLoadingReady )
   END_RUNG
   RUNG wire#w1
      Contact( "Unit1.Em5.ControlNodes".cmTransferPnPLeftClampOpenClose.monitoring.inHomePos )
      Coil( "Unit1.Em5.ControlNodes".GRnR_TransferPnP.jobInterface.transferPnPLeft.hipotThicknessPLACEJob3.unClampDone )
   END_RUNG
   RUNG wire#powerrail
      Contact( "Unit1.Em5.ControlNodes".GRnR_TransferPnP.jobInterface.transferPnPLeft.hipotThicknessPLACEJob3.workingDone )
      wire#w2
      Coil( "Unit1.Em5.ControlNodes".GRnR_TransferPnP.jobInterface.transferPnPLeft.hipotThicknessPLACEJob3.unLoadingDone )
   END_RUNG
   RUNG wire#powerrail
      Contact( #instGRnR_HipotThicknessUnloadJob3_Left.jobStatus.active )
      Contact( "Unit1.Em5.ControlNodes".GRnR_TransferPnP."step".transition1[380] )
   END_RUNG wire#w2
   // the same network as SCL:
   "Unit1.Em5.ControlNodes".GRnR_TransferPnP.jobInterface.transferPnPLeft.hipotThicknessPLACEJob3.unLoadingReady := #instGRnR_HipotThicknessUnloadJob3_Left.jobStatus.active AND "Unit1.Em5.ControlNodes".cm.softcam.transferPnPLeftAxisX.pos04_hipotThickness.inPos AND "Unit1.Em5.ControlNodes".cm.softcam.transferPnPLeftAxisY.pos04_hipotThickness.inPos AND "Unit1.Em5.ControlNodes".cm.softcam.transferPnPLeftAxisZ.pos04_hipotThickness.inPos;
   "Unit1.Em5.ControlNodes".GRnR_TransferPnP.jobInterface.transferPnPLeft.hipotThicknessPLACEJob3.unClampDone := "Unit1.Em5.ControlNodes".GRnR_TransferPnP.jobInterface.transferPnPLeft.hipotThicknessPLACEJob3.unLoadingReady AND "Unit1.Em5.ControlNodes".cmTransferPnPLeftClampOpenClose.monitoring.inHomePos;
   "Unit1.Em5.ControlNodes".GRnR_TransferPnP.jobInterface.transferPnPLeft.hipotThicknessPLACEJob3.unLoadingDone := "Unit1.Em5.ControlNodes".GRnR_TransferPnP.jobInterface.transferPnPLeft.hipotThicknessPLACEJob3.workingDone OR (#instGRnR_HipotThicknessUnloadJob3_Left.jobStatus.active AND "Unit1.Em5.ControlNodes".GRnR_TransferPnP."step".transition1[380]);
END_REGION

REGION Network 64: Transfer P&P Gague R&R Job Interface [Hipot & Thickness Loading][Left]
   RUNG wire#powerrail
      Contact( #instGRnR_HipotThicknessLoadJob4_Left.jobStatus.active )
      Contact( "Unit1.Em5.ControlNodes".cm.softcam.transferPnPLeftAxisX.pos04_hipotThickness.inPos )
      Contact( "Unit1.Em5.ControlNodes".cm.softcam.transferPnPLeftAxisY.pos04_hipotThickness.inPos )
      Contact( "Unit1.Em5.ControlNodes".cm.softcam.transferPnPLeftAxisZ.pos04_hipotThickness.inPos )
      wire#w1
      Coil( "Unit1.Em5.ControlNodes".GRnR_TransferPnP.jobInterface.transferPnPLeft.hipotThicknessPICKJob4.loadingReady )
   END_RUNG
   RUNG wire#w1
      Contact( "Unit1.Em5.ControlNodes".cmTransferPnPLeftClampOpenClose.monitoring.inWorkPos )
      Coil( "Unit1.Em5.ControlNodes".GRnR_TransferPnP.jobInterface.transferPnPLeft.hipotThicknessPICKJob4.clampDone )
   END_RUNG
   RUNG wire#powerrail
      Contact( "Unit1.Em5.ControlNodes".GRnR_TransferPnP.jobInterface.transferPnPLeft.hipotThicknessPICKJob4.workingDone )
      wire#w2
      Coil( "Unit1.Em5.ControlNodes".GRnR_TransferPnP.jobInterface.transferPnPLeft.hipotThicknessPICKJob4.loadingDone )
   END_RUNG
   RUNG wire#powerrail
      Contact( #instGRnR_HipotThicknessLoadJob4_Left.jobStatus.active )
      Contact( "Unit1.Em5.ControlNodes".GRnR_TransferPnP."step".transition1[480] )
   END_RUNG wire#w2
   // the same network as SCL:
   "Unit1.Em5.ControlNodes".GRnR_TransferPnP.jobInterface.transferPnPLeft.hipotThicknessPICKJob4.loadingReady := #instGRnR_HipotThicknessLoadJob4_Left.jobStatus.active AND "Unit1.Em5.ControlNodes".cm.softcam.transferPnPLeftAxisX.pos04_hipotThickness.inPos AND "Unit1.Em5.ControlNodes".cm.softcam.transferPnPLeftAxisY.pos04_hipotThickness.inPos AND "Unit1.Em5.ControlNodes".cm.softcam.transferPnPLeftAxisZ.pos04_hipotThickness.inPos;
   "Unit1.Em5.ControlNodes".GRnR_TransferPnP.jobInterface.transferPnPLeft.hipotThicknessPICKJob4.clampDone := "Unit1.Em5.ControlNodes".GRnR_TransferPnP.jobInterface.transferPnPLeft.hipotThicknessPICKJob4.loadingReady AND "Unit1.Em5.ControlNodes".cmTransferPnPLeftClampOpenClose.monitoring.inWorkPos;
   "Unit1.Em5.ControlNodes".GRnR_TransferPnP.jobInterface.transferPnPLeft.hipotThicknessPICKJob4.loadingDone := "Unit1.Em5.ControlNodes".GRnR_TransferPnP.jobInterface.transferPnPLeft.hipotThicknessPICKJob4.workingDone OR (#instGRnR_HipotThicknessLoadJob4_Left.jobStatus.active AND "Unit1.Em5.ControlNodes".GRnR_TransferPnP."step".transition1[480]);
END_REGION

